;bead-perimeter_outer
$VEL.CP=1
LIN {X -65.721,Y -278.478,Z 40.000,A 0.000,B 0.000,C 180.000,E1 0.000} C_DIS
LIN {X -51.297,Y -281.492,Z 40.000,A 0.000,B 0.000,C 180.000,E1 0.000} C_DIS
LIN {X -36.738,Y -283.759,Z 40.000,A 0.000,B 0.000,C 180.000,E1 0.000} C_DIS
LIN {X -22.082,Y -285.274,Z 40.000,A 0.000,B 0.000,C 180.000,E1 0.000} C_DIS
LIN {X -7.367,Y -286.033,Z 40.000,A 0.000,B 0.000,C 180.000,E1 0.000} C_DIS
LIN {X 7.367,Y -286.033,Z 40.000,A 0.000,B 0.000,C 180.000,E1 0.000} C_DIS
LIN {X 16.843,Y -285.545,Z 40.000,A 0.000,B 0.000,C 180.000,E1 0.000} C_DIS
LIN {X 22.082,Y -285.274,Z 40.000,A 0.000,B 0.000,C 180.000,E1 0.000} C_DIS
LIN {X 36.738,Y -283.759,Z 40.000,A 0.000,B 0.000,C 180.000,E1 0.000} C_DIS
LIN {X 51.297,Y -281.492,Z 40.000,A 0.000,B 0.000,C 180.000,E1 0.000} C_DIS
LIN {X 65.721,Y -278.478,Z 40.000,A 0.000,B 0.000,C 180.000,E1 0.000} C_DIS
LIN {X 79.969,Y -274.726,Z 40.000,A 0.000,B 0.000,C 180.000,E1 0.000} C_DIS
LIN {X 94.005,Y -270.245,Z 40.000,A 0.000,B 0.000,C 180.000,E1 0.000} C_DIS
LIN {X 107.792,Y -265.047,Z 40.000,A 0.000,B 0.000,C 180.000,E1 0.000} C_DIS
LIN {X 121.294,Y -259.146,Z 40.000,A 0.000,B 0.000,C 180.000,E1 0.000} C_DIS
LIN {X 134.474,Y -252.559,Z 40.000,A 0.000,B 0.000,C 180.000,E1 0.000} C_DIS
LIN {X 147.297,Y -245.302,Z 40.000,A 0.000,B 0.000,C 180.000,E1 0.000} C_DIS
LIN {X 159.730,Y -237.393,Z 40.000,A 0.000,B 0.000,C 180.000,E1 0.000} C_DIS
LIN {X 171.739,Y -228.857,Z 40.000,A 0.000,B 0.000,C 180.000,E1 0.000} C_DIS
LIN {X 183.292,Y -219.713,Z 40.000,A 0.000,B 0.000,C 180.000,E1 0.000} C_DIS
LIN {X 194.358,Y -209.985,Z 40.000,A 0.000,B 0.000,C 180.000,E1 0.000} C_DIS
LIN {X 204.911,Y -199.701,Z 40.000,A 0.000,B 0.000,C 180.000,E1 0.000} C_DIS
LIN {X 214.920,Y -188.888,Z 40.000,A 0.000,B 0.000,C 180.000,E1 0.000} C_DIS
LIN {X 224.358,Y -177.574,Z 40.000,A 0.000,B 0.000,C 180.000,E1 0.000} C_DIS
LIN {X 233.202,Y -165.788,Z 40.000,A 0.000,B 0.000,C 180.000,E1 0.000} C_DIS
LIN {X 241.428,Y -153.563,Z 40.000,A 0.000,B 0.000,C 180.000,E1 0.000} C_DIS
LIN {X 249.014,Y -140.932,Z 40.000,A 0.000,B 0.000,C 180.000,E1 0.000} C_DIS
LIN {X 255.938,Y -127.926,Z 40.000,A 0.000,B 0.000,C 180.000,E1 0.000} C_DIS
LIN {X 262.185,Y -114.581,Z 40.000,A 0.000,B 0.000,C 180.000,E1 0.000} C_DIS
LIN {X 267.735,Y -100.933,Z 40.000,A 0.000,B 0.000,C 180.000,E1 0.000} C_DIS
LIN {X 272.575,Y -87.015,Z 40.000,A 0.000,B 0.000,C 180.000,E1 0.000} C_DIS
LIN {X 276.694,Y -72.868,Z 40.000,A 0.000,B 0.000,C 180.000,E1 0.000} C_DIS
LIN {X 280.078,Y -58.528,Z 40.000,A 0.000,B 0.000,C 180.000,E1 0.000} C_DIS
LIN {X 282.720,Y -44.032,Z 40.000,A 0.000,B 0.000,C 180.000,E1 0.000} C_DIS
LIN {X 284.612,Y -29.420,Z 40.000,A 0.000,B 0.000,C 180.000,E1 0.000} C_DIS
LIN {X 285.749,Y -14.730,Z 40.000,A 0.000,B 0.000,C 180.000,E1 0.000} C_DIS
LIN {X 286.128,Y 0.000,Z 40.000,A 0.000,B 0.000,C 180.000,E1 0.000} C_DIS
LIN {X 285.749,Y 14.730,Z 40.000,A 0.000,B 0.000,C 180.000,E1 0.000} C_DIS
LIN {X 284.612,Y 29.420,Z 40.000,A 0.000,B 0.000,C 180.000,E1 0.000} C_DIS
LIN {X 282.720,Y 44.032,Z 40.000,A 0.000,B 0.000,C 180.000,E1 0.000} C_DIS
LIN {X 280.078,Y 58.528,Z 40.000,A 0.000,B 0.000,C 180.000,E1 0.000} C_DIS
LIN {X 276.694,Y 72.868,Z 40.000,A 0.000,B 0.000,C 180.000,E1 0.000} C_DIS
LIN {X 272.575,Y 87.015,Z 40.000,A 0.000,B 0.000,C 180.000,E1 0.000} C_DIS
LIN {X 267.735,Y 100.932,Z 40.000,A 0.000,B 0.000,C 180.000,E1 0.000} C_DIS
LIN {X 262.185,Y 114.581,Z 40.000,A 0.000,B 0.000,C 180.000,E1 0.000} C_DIS
LIN {X 255.938,Y 127.926,Z 40.000,A 0.000,B 0.000,C 180.000,E1 0.000} C_DIS
LIN {X 249.014,Y 140.932,Z 40.000,A 0.000,B 0.000,C 180.000,E1 0.000} C_DIS
LIN {X 241.428,Y 153.563,Z 40.000,A 0.000,B 0.000,C 180.000,E1 0.000} C_DIS
LIN {X 233.202,Y 165.788,Z 40.000,A 0.000,B 0.000,C 180.000,E1 0.000} C_DIS
LIN {X 224.358,Y 177.574,Z 40.000,A 0.000,B 0.000,C 180.000,E1 0.000} C_DIS
LIN {X 214.920,Y 188.888,Z 40.000,A 0.000,B 0.000,C 180.000,E1 0.000} C_DIS
LIN {X 204.911,Y 199.701,Z 40.000,A 0.000,B 0.000,C 180.000,E1 0.000} C_DIS
LIN {X 194.358,Y 209.985,Z 40.000,A 0.000,B 0.000,C 180.000,E1 0.000} C_DIS
LIN {X 183.292,Y 219.713,Z 40.000,A 0.000,B 0.000,C 180.000,E1 0.000} C_DIS
LIN {X 171.739,Y 228.857,Z 40.000,A 0.000,B 0.000,C 180.000,E1 0.000} C_DIS
LIN {X 159.730,Y 237.393,Z 40.000,A 0.000,B 0.000,C 180.000,E1 0.000} C_DIS
LIN {X 147.297,Y 245.302,Z 40.000,A 0.000,B 0.000,C 180.000,E1 0.000} C_DIS
LIN {X 134.474,Y 252.559,Z 40.000,A 0.000,B 0.000,C 180.000,E1 0.000} C_DIS
LIN {X 121.294,Y 259.146,Z 40.000,A 0.000,B 0.000,C 180.000,E1 0.000} C_DIS
LIN {X 107.792,Y 265.047,Z 40.000,A 0.000,B 0.000,C 180.000,E1 0.000} C_DIS
LIN {X 94.005,Y 270.245,Z 40.000,A 0.000,B 0.000,C 180.000,E1 0.000} C_DIS
LIN {X 79.969,Y 274.726,Z 40.000,A 0.000,B 0.000,C 180.000,E1 0.000} C_DIS
LIN {X 65.721,Y 278.478,Z 40.000,A 0.000,B 0.000,C 180.000,E1 0.000} C_DIS
LIN {X 51.297,Y 281.492,Z 40.000,A 0.000,B 0.000,C 180.000,E1 0.000} C_DIS
LIN {X 36.738,Y 283.759,Z 40.000,A 0.000,B 0.000,C 180.000,E1 0.000} C_DIS
LIN {X 22.082,Y 285.274,Z 40.000,A 0.000,B 0.000,C 180.000,E1 0.000} C_DIS
LIN {X 7.367,Y 286.033,Z 40.000,A 0.000,B 0.000,C 180.000,E1 0.000} C_DIS
LIN {X -7.367,Y 286.033,Z 40.000,A 0.000,B 0.000,C 180.000,E1 0.000} C_DIS
LIN {X -22.082,Y 285.274,Z 40.000,A 0.000,B 0.000,C 180.000,E1 0.000} C_DIS
LIN {X -36.738,Y 283.759,Z 40.000,A 0.000,B 0.000,C 180.000,E1 0.000} C_DIS
LIN {X -51.297,Y 281.492,Z 40.000,A 0.000,B 0.000,C 180.000,E1 0.000} C_DIS
LIN {X -65.721,Y 278.478,Z 40.000,A 0.000,B 0.000,C 180.000,E1 0.000} C_DIS
LIN {X -79.969,Y 274.726,Z 40.000,A 0.000,B 0.000,C 180.000,E1 0.000} C_DIS
LIN {X -94.005,Y 270.245,Z 40.000,A 0.000,B 0.000,C 180.000,E1 0.000} C_DIS
LIN {X -107.792,Y 265.047,Z 40.000,A 0.000,B 0.000,C 180.000,E1 0.000} C_DIS
LIN {X -121.294,Y 259.146,Z 40.000,A 0.000,B 0.000,C 180.000,E1 0.000} C_DIS
LIN {X -134.474,Y 252.559,Z 40.000,A 0.000,B 0.000,C 180.000,E1 0.000} C_DIS
LIN {X -147.297,Y 245.302,Z 40.000,A 0.000,B 0.000,C 180.000,E1 0.000} C_DIS
LIN {X -159.730,Y 237.393,Z 40.000,A 0.000,B 0.000,C 180.000,E1 0.000} C_DIS
LIN {X -171.739,Y 228.857,Z 40.000,A 0.000,B 0.000,C 180.000,E1 0.000} C_DIS
LIN {X -183.292,Y 219.713,Z 40.000,A 0.000,B 0.000,C 180.000,E1 0.000} C_DIS
LIN {X -194.358,Y 209.985,Z 40.000,A 0.000,B 0.000,C 180.000,E1 0.000} C_DIS
LIN {X -204.911,Y 199.701,Z 40.000,A 0.000,B 0.000,C 180.000,E1 0.000} C_DIS
LIN {X -214.920,Y 188.888,Z 40.000,A 0.000,B 0.000,C 180.000,E1 0.000} C_DIS
LIN {X -224.358,Y 177.574,Z 40.000,A 0.000,B 0.000,C 180.000,E1 0.000} C_DIS
LIN {X -233.202,Y 165.788,Z 40.000,A 0.000,B 0.000,C 180.000,E1 0.000} C_DIS
LIN {X -241.428,Y 153.563,Z 40.000,A 0.000,B 0.000,C 180.000,E1 0.000} C_DIS
LIN {X -249.014,Y 140.932,Z 40.000,A 0.000,B 0.000,C 180.000,E1 0.000} C_DIS
LIN {X -255.938,Y 127.926,Z 40.000,A 0.000,B 0.000,C 180.000,E1 0.000} C_DIS
LIN {X -262.185,Y 114.581,Z 40.000,A 0.000,B 0.000,C 180.000,E1 0.000} C_DIS
LIN {X -267.735,Y 100.933,Z 40.000,A 0.000,B 0.000,C 180.000,E1 0.000} C_DIS
LIN {X -272.575,Y 87.015,Z 40.000,A 0.000,B 0.000,C 180.000,E1 0.000} C_DIS
LIN {X -276.694,Y 72.868,Z 40.000,A 0.000,B 0.000,C 180.000,E1 0.000} C_DIS
LIN {X -280.078,Y 58.528,Z 40.000,A 0.000,B 0.000,C 180.000,E1 0.000} C_DIS
LIN {X -282.720,Y 44.032,Z 40.000,A 0.000,B 0.000,C 180.000,E1 0.000} C_DIS
LIN {X -284.612,Y 29.420,Z 40.000,A 0.000,B 0.000,C 180.000,E1 0.000} C_DIS
LIN {X -285.749,Y 14.730,Z 40.000,A 0.000,B 0.000,C 180.000,E1 0.000} C_DIS
LIN {X -286.128,Y 0.000,Z 40.000,A 0.000,B 0.000,C 180.000,E1 0.000} C_DIS
LIN {X -285.749,Y -14.730,Z 40.000,A 0.000,B 0.000,C 180.000,E1 0.000} C_DIS
LIN {X -284.612,Y -29.420,Z 40.000,A 0.000,B 0.000,C 180.000,E1 0.000} C_DIS
LIN {X -282.720,Y -44.032,Z 40.000,A 0.000,B 0.000,C 180.000,E1 0.000} C_DIS
LIN {X -280.078,Y -58.528,Z 40.000,A 0.000,B 0.000,C 180.000,E1 0.000} C_DIS
LIN {X -276.694,Y -72.868,Z 40.000,A 0.000,B 0.000,C 180.000,E1 0.000} C_DIS
LIN {X -272.575,Y -87.015,Z 40.000,A 0.000,B 0.000,C 180.000,E1 0.000} C_DIS
LIN {X -269.459,Y -95.976,Z 40.000,A 0.000,B 0.000,C 180.000,E1 0.000} C_DIS
LIN {X -267.735,Y -100.932,Z 40.000,A 0.000,B 0.000,C 180.000,E1 0.000} C_DIS
LIN {X -262.185,Y -114.581,Z 40.000,A 0.000,B 0.000,C 180.000,E1 0.000} C_DIS
LIN {X -255.938,Y -127.926,Z 40.000,A 0.000,B 0.000,C 180.000,E1 0.000} C_DIS
LIN {X -249.014,Y -140.932,Z 40.000,A 0.000,B 0.000,C 180.000,E1 0.000} C_DIS
LIN {X -241.428,Y -153.563,Z 40.000,A 0.000,B 0.000,C 180.000,E1 0.000} C_DIS
LIN {X -233.202,Y -165.788,Z 40.000,A 0.000,B 0.000,C 180.000,E1 0.000} C_DIS
LIN {X -224.358,Y -177.574,Z 40.000,A 0.000,B 0.000,C 180.000,E1 0.000} C_DIS
LIN {X -214.920,Y -188.888,Z 40.000,A 0.000,B 0.000,C 180.000,E1 0.000} C_DIS
LIN {X -204.911,Y -199.701,Z 40.000,A 0.000,B 0.000,C 180.000,E1 0.000} C_DIS
LIN {X -194.358,Y -209.985,Z 40.000,A 0.000,B 0.000,C 180.000,E1 0.000} C_DIS
LIN {X -183.292,Y -219.713,Z 40.000,A 0.000,B 0.000,C 180.000,E1 0.000} C_DIS
LIN {X -171.739,Y -228.857,Z 40.000,A 0.000,B 0.000,C 180.000,E1 0.000} C_DIS
LIN {X -159.730,Y -237.393,Z 40.000,A 0.000,B 0.000,C 180.000,E1 0.000} C_DIS
LIN {X -147.297,Y -245.302,Z 40.000,A 0.000,B 0.000,C 180.000,E1 0.000} C_DIS
LIN {X -134.474,Y -252.559,Z 40.000,A 0.000,B 0.000,C 180.000,E1 0.000} C_DIS
LIN {X -121.294,Y -259.146,Z 40.000,A 0.000,B 0.000,C 180.000,E1 0.000} C_DIS
LIN {X -107.792,Y -265.047,Z 40.000,A 0.000,B 0.000,C 180.000,E1 0.000} C_DIS
LIN {X -94.005,Y -270.245,Z 40.000,A 0.000,B 0.000,C 180.000,E1 0.000} C_DIS
LIN {X -79.969,Y -274.726,Z 40.000,A 0.000,B 0.000,C 180.000,E1 0.000} C_DIS
;rapid-leaky
$VEL.CP=0.3
LIN {X -75.624,Y -259.800,Z 40.000,A 0.000,B 0.000,C 180.000,E1 0.000} C_DIS
;bead-perimeter_inner
$VEL.CP=1
LIN {X -62.150,Y -263.349,Z 40.000,A 0.000,B 0.000,C 180.000,E1 0.000} C_DIS
LIN {X -48.511,Y -266.199,Z 40.000,A 0.000,B 0.000,C 180.000,E1 0.000} C_DIS
LIN {X -34.743,Y -268.343,Z 40.000,A 0.000,B 0.000,C 180.000,E1 0.000} C_DIS
LIN {X -20.882,Y -269.776,Z 40.000,A 0.000,B 0.000,C 180.000,E1 0.000} C_DIS
LIN {X -6.967,Y -270.493,Z 40.000,A 0.000,B 0.000,C 180.000,E1 0.000} C_DIS
LIN {X 6.967,Y -270.493,Z 40.000,A 0.000,B 0.000,C 180.000,E1 0.000} C_DIS
LIN {X 16.043,Y -270.025,Z 40.000,A 0.000,B 0.000,C 180.000,E1 0.000} C_DIS
LIN {X 20.882,Y -269.776,Z 40.000,A 0.000,B 0.000,C 180.000,E1 0.000} C_DIS
LIN {X 34.743,Y -268.343,Z 40.000,A 0.000,B 0.000,C 180.000,E1 0.000} C_DIS
LIN {X 48.511,Y -266.199,Z 40.000,A 0.000,B 0.000,C 180.000,E1 0.000} C_DIS
LIN {X 62.150,Y -263.349,Z 40.000,A 0.000,B 0.000,C 180.000,E1 0.000} C_DIS
LIN {X 75.624,Y -259.800,Z 40.000,A 0.000,B 0.000,C 180.000,E1 0.000} C_DIS
LIN {X 88.898,Y -255.563,Z 40.000,A 0.000,B 0.000,C 180.000,E1 0.000} C_DIS
LIN {X 101.936,Y -250.648,Z 40.000,A 0.000,B 0.000,C 180.000,E1 0.000} C_DIS
LIN {X 114.704,Y -245.067,Z 40.000,A 0.000,B 0.000,C 180.000,E1 0.000} C_DIS
LIN {X 127.168,Y -238.838,Z 40.000,A 0.000,B 0.000,C 180.000,E1 0.000} C_DIS
LIN {X 139.294,Y -231.975,Z 40.000,A 0.000,B 0.000,C 180.000,E1 0.000} C_DIS
LIN {X 151.052,Y -224.496,Z 40.000,A 0.000,B 0.000,C 180.000,E1 0.000} C_DIS
LIN {X 162.409,Y -216.423,Z 40.000,A 0.000,B 0.000,C 180.000,E1 0.000} C_DIS
LIN {X 173.333,Y -207.776,Z 40.000,A 0.000,B 0.000,C 180.000,E1 0.000} C_DIS
LIN {X 183.799,Y -198.577,Z 40.000,A 0.000,B 0.000,C 180.000,E1 0.000} C_DIS
LIN {X 193.778,Y -188.852,Z 40.000,A 0.000,B 0.000,C 180.000,E1 0.000} C_DIS
LIN {X 203.243,Y -178.626,Z 40.000,A 0.000,B 0.000,C 180.000,E1 0.000} C_DIS
LIN {X 212.169,Y -167.927,Z 40.000,A 0.000,B 0.000,C 180.000,E1 0.000} C_DIS
LIN {X 220.533,Y -156.781,Z 40.000,A 0.000,B 0.000,C 180.000,E1 0.000} C_DIS
LIN {X 228.312,Y -145.220,Z 40.000,A 0.000,B 0.000,C 180.000,E1 0.000} C_DIS
LIN {X 235.485,Y -133.275,Z 40.000,A 0.000,B 0.000,C 180.000,E1 0.000} C_DIS
LIN {X 242.033,Y -120.975,Z 40.000,A 0.000,B 0.000,C 180.000,E1 0.000} C_DIS
LIN {X 247.940,Y -108.356,Z 40.000,A 0.000,B 0.000,C 180.000,E1 0.000} C_DIS
LIN {X 253.189,Y -95.450,Z 40.000,A 0.000,B 0.000,C 180.000,E1 0.000} C_DIS
LIN {X 257.767,Y -82.287,Z 40.000,A 0.000,B 0.000,C 180.000,E1 0.000} C_DIS
LIN {X 261.662,Y -68.909,Z 40.000,A 0.000,B 0.000,C 180.000,E1 0.000} C_DIS
LIN {X 264.862,Y -55.348,Z 40.000,A 0.000,B 0.000,C 180.000,E1 0.000} C_DIS
LIN {X 267.360,Y -41.639,Z 40.000,A 0.000,B 0.000,C 180.000,E1 0.000} C_DIS
LIN {X 269.149,Y -27.822,Z 40.000,A 0.000,B 0.000,C 180.000,E1 0.000} C_DIS
LIN {X 270.224,Y -13.929,Z 40.000,A 0.000,B 0.000,C 180.000,E1 0.000} C_DIS
LIN {X 270.583,Y 0.000,Z 40.000,A 0.000,B 0.000,C 180.000,E1 0.000} C_DIS
LIN {X 270.224,Y 13.929,Z 40.000,A 0.000,B 0.000,C 180.000,E1 0.000} C_DIS
LIN {X 269.149,Y 27.822,Z 40.000,A 0.000,B 0.000,C 180.000,E1 0.000} C_DIS
LIN {X 267.360,Y 41.639,Z 40.000,A 0.000,B 0.000,C 180.000,E1 0.000} C_DIS
LIN {X 264.862,Y 55.348,Z 40.000,A 0.000,B 0.000,C 180.000,E1 0.000} C_DIS
LIN {X 261.662,Y 68.909,Z 40.000,A 0.000,B 0.000,C 180.000,E1 0.000} C_DIS
LIN {X 257.766,Y 82.288,Z 40.000,A 0.000,B 0.000,C 180.000,E1 0.000} C_DIS
LIN {X 253.189,Y 95.449,Z 40.000,A 0.000,B 0.000,C 180.000,E1 0.000} C_DIS
LIN {X 247.940,Y 108.356,Z 40.000,A 0.000,B 0.000,C 180.000,E1 0.000} C_DIS
LIN {X 242.033,Y 120.975,Z 40.000,A 0.000,B 0.000,C 180.000,E1 0.000} C_DIS
LIN {X 235.485,Y 133.275,Z 40.000,A 0.000,B 0.000,C 180.000,E1 0.000} C_DIS
LIN {X 228.312,Y 145.220,Z 40.000,A 0.000,B 0.000,C 180.000,E1 0.000} C_DIS
LIN {X 220.533,Y 156.781,Z 40.000,A 0.000,B 0.000,C 180.000,E1 0.000} C_DIS
LIN {X 212.169,Y 167.927,Z 40.000,A 0.000,B 0.000,C 180.000,E1 0.000} C_DIS
LIN {X 203.243,Y 178.626,Z 40.000,A 0.000,B 0.000,C 180.000,E1 0.000} C_DIS
LIN {X 193.778,Y 188.852,Z 40.000,A 0.000,B 0.000,C 180.000,E1 0.000} C_DIS
LIN {X 183.799,Y 198.577,Z 40.000,A 0.000,B 0.000,C 180.000,E1 0.000} C_DIS
LIN {X 173.333,Y 207.776,Z 40.000,A 0.000,B 0.000,C 180.000,E1 0.000} C_DIS
LIN {X 162.409,Y 216.423,Z 40.000,A 0.000,B 0.000,C 180.000,E1 0.000} C_DIS
LIN {X 151.052,Y 224.496,Z 40.000,A 0.000,B 0.000,C 180.000,E1 0.000} C_DIS
LIN {X 139.294,Y 231.975,Z 40.000,A 0.000,B 0.000,C 180.000,E1 0.000} C_DIS
LIN {X 127.168,Y 238.838,Z 40.000,A 0.000,B 0.000,C 180.000,E1 0.000} C_DIS
LIN {X 114.704,Y 245.067,Z 40.000,A 0.000,B 0.000,C 180.000,E1 0.000} C_DIS
LIN {X 101.936,Y 250.648,Z 40.000,A 0.000,B 0.000,C 180.000,E1 0.000} C_DIS
LIN {X 88.898,Y 255.563,Z 40.000,A 0.000,B 0.000,C 180.000,E1 0.000} C_DIS
LIN {X 75.624,Y 259.800,Z 40.000,A 0.000,B 0.000,C 180.000,E1 0.000} C_DIS
LIN {X 62.150,Y 263.349,Z 40.000,A 0.000,B 0.000,C 180.000,E1 0.000} C_DIS
LIN {X 48.511,Y 266.199,Z 40.000,A 0.000,B 0.000,C 180.000,E1 0.000} C_DIS
LIN {X 34.743,Y 268.343,Z 40.000,A 0.000,B 0.000,C 180.000,E1 0.000} C_DIS
LIN {X 20.882,Y 269.776,Z 40.000,A 0.000,B 0.000,C 180.000,E1 0.000} C_DIS
LIN {X 6.967,Y 270.493,Z 40.000,A 0.000,B 0.000,C 180.000,E1 0.000} C_DIS
LIN {X -6.967,Y 270.493,Z 40.000,A 0.000,B 0.000,C 180.000,E1 0.000} C_DIS
LIN {X -20.882,Y 269.776,Z 40.000,A 0.000,B 0.000,C 180.000,E1 0.000} C_DIS
LIN {X -34.743,Y 268.343,Z 40.000,A 0.000,B 0.000,C 180.000,E1 0.000} C_DIS
LIN {X -48.511,Y 266.199,Z 40.000,A 0.000,B 0.000,C 180.000,E1 0.000} C_DIS
LIN {X -62.150,Y 263.349,Z 40.000,A 0.000,B 0.000,C 180.000,E1 0.000} C_DIS
LIN {X -75.624,Y 259.800,Z 40.000,A 0.000,B 0.000,C 180.000,E1 0.000} C_DIS
LIN {X -88.898,Y 255.563,Z 40.000,A 0.000,B 0.000,C 180.000,E1 0.000} C_DIS
LIN {X -101.936,Y 250.648,Z 40.000,A 0.000,B 0.000,C 180.000,E1 0.000} C_DIS
LIN {X -114.704,Y 245.067,Z 40.000,A 0.000,B 0.000,C 180.000,E1 0.000} C_DIS
LIN {X -127.168,Y 238.838,Z 40.000,A 0.000,B 0.000,C 180.000,E1 0.000} C_DIS
LIN {X -139.294,Y 231.975,Z 40.000,A 0.000,B 0.000,C 180.000,E1 0.000} C_DIS
LIN {X -151.052,Y 224.496,Z 40.000,A 0.000,B 0.000,C 180.000,E1 0.000} C_DIS
LIN {X -162.409,Y 216.423,Z 40.000,A 0.000,B 0.000,C 180.000,E1 0.000} C_DIS
LIN {X -173.333,Y 207.776,Z 40.000,A 0.000,B 0.000,C 180.000,E1 0.000} C_DIS
LIN {X -183.799,Y 198.577,Z 40.000,A 0.000,B 0.000,C 180.000,E1 0.000} C_DIS
LIN {X -193.778,Y 188.852,Z 40.000,A 0.000,B 0.000,C 180.000,E1 0.000} C_DIS
LIN {X -203.243,Y 178.626,Z 40.000,A 0.000,B 0.000,C 180.000,E1 0.000} C_DIS
LIN {X -212.169,Y 167.927,Z 40.000,A 0.000,B 0.000,C 180.000,E1 0.000} C_DIS
LIN {X -220.533,Y 156.781,Z 40.000,A 0.000,B 0.000,C 180.000,E1 0.000} C_DIS
LIN {X -228.312,Y 145.220,Z 40.000,A 0.000,B 0.000,C 180.000,E1 0.000} C_DIS
LIN {X -235.485,Y 133.275,Z 40.000,A 0.000,B 0.000,C 180.000,E1 0.000} C_DIS
LIN {X -242.033,Y 120.975,Z 40.000,A 0.000,B 0.000,C 180.000,E1 0.000} C_DIS
LIN {X -247.940,Y 108.356,Z 40.000,A 0.000,B 0.000,C 180.000,E1 0.000} C_DIS
LIN {X -253.189,Y 95.450,Z 40.000,A 0.000,B 0.000,C 180.000,E1 0.000} C_DIS
LIN {X -257.767,Y 82.287,Z 40.000,A 0.000,B 0.000,C 180.000,E1 0.000} C_DIS
LIN {X -261.662,Y 68.909,Z 40.000,A 0.000,B 0.000,C 180.000,E1 0.000} C_DIS
LIN {X -264.862,Y 55.348,Z 40.000,A 0.000,B 0.000,C 180.000,E1 0.000} C_DIS
LIN {X -267.360,Y 41.639,Z 40.000,A 0.000,B 0.000,C 180.000,E1 0.000} C_DIS
LIN {X -269.149,Y 27.822,Z 40.000,A 0.000,B 0.000,C 180.000,E1 0.000} C_DIS
LIN {X -270.224,Y 13.929,Z 40.000,A 0.000,B 0.000,C 180.000,E1 0.000} C_DIS
LIN {X -270.583,Y 0.000,Z 40.000,A 0.000,B 0.000,C 180.000,E1 0.000} C_DIS
LIN {X -270.224,Y -13.929,Z 40.000,A 0.000,B 0.000,C 180.000,E1 0.000} C_DIS
LIN {X -269.149,Y -27.822,Z 40.000,A 0.000,B 0.000,C 180.000,E1 0.000} C_DIS
LIN {X -267.360,Y -41.639,Z 40.000,A 0.000,B 0.000,C 180.000,E1 0.000} C_DIS
LIN {X -264.862,Y -55.348,Z 40.000,A 0.000,B 0.000,C 180.000,E1 0.000} C_DIS
LIN {X -261.662,Y -68.909,Z 40.000,A 0.000,B 0.000,C 180.000,E1 0.000} C_DIS
LIN {X -257.766,Y -82.288,Z 40.000,A 0.000,B 0.000,C 180.000,E1 0.000} C_DIS
LIN {X -254.782,Y -90.870,Z 40.000,A 0.000,B 0.000,C 180.000,E1 0.000} C_DIS
LIN {X -253.189,Y -95.449,Z 40.000,A 0.000,B 0.000,C 180.000,E1 0.000} C_DIS
LIN {X -247.940,Y -108.356,Z 40.000,A 0.000,B 0.000,C 180.000,E1 0.000} C_DIS
LIN {X -242.033,Y -120.975,Z 40.000,A 0.000,B 0.000,C 180.000,E1 0.000} C_DIS
LIN {X -235.485,Y -133.275,Z 40.000,A 0.000,B 0.000,C 180.000,E1 0.000} C_DIS
LIN {X -228.312,Y -145.220,Z 40.000,A 0.000,B 0.000,C 180.000,E1 0.000} C_DIS
LIN {X -220.533,Y -156.781,Z 40.000,A 0.000,B 0.000,C 180.000,E1 0.000} C_DIS
LIN {X -212.169,Y -167.927,Z 40.000,A 0.000,B 0.000,C 180.000,E1 0.000} C_DIS
LIN {X -203.243,Y -178.626,Z 40.000,A 0.000,B 0.000,C 180.000,E1 0.000} C_DIS
LIN {X -193.778,Y -188.852,Z 40.000,A 0.000,B 0.000,C 180.000,E1 0.000} C_DIS
LIN {X -183.799,Y -198.577,Z 40.000,A 0.000,B 0.000,C 180.000,E1 0.000} C_DIS
LIN {X -173.333,Y -207.776,Z 40.000,A 0.000,B 0.000,C 180.000,E1 0.000} C_DIS
LIN {X -162.409,Y -216.423,Z 40.000,A 0.000,B 0.000,C 180.000,E1 0.000} C_DIS
LIN {X -151.052,Y -224.496,Z 40.000,A 0.000,B 0.000,C 180.000,E1 0.000} C_DIS
LIN {X -139.294,Y -231.975,Z 40.000,A 0.000,B 0.000,C 180.000,E1 0.000} C_DIS
LIN {X -127.168,Y -238.838,Z 40.000,A 0.000,B 0.000,C 180.000,E1 0.000} C_DIS
LIN {X -114.704,Y -245.067,Z 40.000,A 0.000,B 0.000,C 180.000,E1 0.000} C_DIS
LIN {X -101.936,Y -250.648,Z 40.000,A 0.000,B 0.000,C 180.000,E1 0.000} C_DIS
LIN {X -88.898,Y -255.563,Z 40.000,A 0.000,B 0.000,C 180.000,E1 0.000} C_DIS
LIN {X -75.624,Y -259.800,Z 40.000,A 0.000,B 0.000,C 180.000,E1 0.000} C_DIS
$VEL.CP=0.3
LIN {X -75.624,Y -259.800,Z 40.000,A 0.000,B 0.000,C 180.000,E1 0.000} C_DIS

EXTRUDER_STATE=FALSE

LIN {X 316.392,Y -180.278,Z 440.000,A 0.000,B 0.000,C 180.000,E1 0.000} C_DIS
LIN {X 126.528,Y -218.793,Z 440.000,A 0.000,B 0.000,C 180.000,E1 0.000} C_DIS
LIN {X 126.528,Y -218.793,Z 40.000,A 0.000,B 0.000,C 180.000,E1 0.000} C_DIS
LIN {X 126.528,Y -218.793,Z 40.000,A 0.000,B 0.000,C 180.000,E1 0.000} C_DIS
EXTRUDER_STATE=TRUE

;bead-solid_infill
$VEL.CP=1
LIN {X 218.862,Y -126.458,Z 40.000,A 0.000,B 0.000,C 180.000,E1 0.000} C_DIS
LIN {X 220.023,Y -124.525,Z 40.000,A 0.000,B 0.000,C 180.000,E1 0.000} C_DIS
LIN {X 222.894,Y -119.132,Z 40.000,A 0.000,B 0.000,C 180.000,E1 0.000} C_DIS
LIN {X 226.142,Y -113.032,Z 40.000,A 0.000,B 0.000,C 180.000,E1 0.000} C_DIS
LIN {X 231.661,Y -101.241,Z 40.000,A 0.000,B 0.000,C 180.000,E1 0.000} C_DIS
LIN {X 236.565,Y -89.183,Z 40.000,A 0.000,B 0.000,C 180.000,E1 0.000} C_DIS
LIN {X 240.842,Y -76.884,Z 40.000,A 0.000,B 0.000,C 180.000,E1 0.000} C_DIS
LIN {X 242.404,Y -71.521,Z 40.000,A 0.000,B 0.000,C 180.000,E1 0.000} C_DIS
LIN {X 71.429,Y -242.496,Z 40.000,A 0.000,B 0.000,C 180.000,E1 0.000} C_DIS
LIN {X 70.658,Y -242.742,Z 40.000,A 0.000,B 0.000,C 180.000,E1 0.000} C_DIS
LIN {X 58.069,Y -246.058,Z 40.000,A 0.000,B 0.000,C 180.000,E1 0.000} C_DIS
LIN {X 45.326,Y -248.721,Z 40.000,A 0.000,B 0.000,C 180.000,E1 0.000} C_DIS
LIN {X 32.462,Y -250.724,Z 40.000,A 0.000,B 0.000,C 180.000,E1 0.000} C_DIS
LIN {X 31.730,Y -250.800,Z 40.000,A 0.000,B 0.000,C 180.000,E1 0.000} C_DIS
LIN {X 250.725,Y -31.804,Z 40.000,A 0.000,B 0.000,C 180.000,E1 0.000} C_DIS
LIN {X 251.478,Y -25.994,Z 40.000,A 0.000,B 0.000,C 180.000,E1 0.000} C_DIS
LIN {X 252.482,Y -13.015,Z 40.000,A 0.000,B 0.000,C 180.000,E1 0.000} C_DIS
LIN {X 252.817,Y 0.000,Z 40.000,A 0.000,B 0.000,C 180.000,E1 0.000} C_DIS
LIN {X 252.775,Y 1.641,Z 40.000,A 0.000,B 0.000,C 180.000,E1 0.000} C_DIS
LIN {X -1.599,Y -252.733,Z 40.000,A 0.000,B 0.000,C 180.000,E1 0.000} C_DIS
LIN {X -6.509,Y -252.733,Z 40.000,A 0.000,B 0.000,C 180.000,E1 0.000} C_DIS
LIN {X -19.511,Y -252.063,Z 40.000,A 0.000,B 0.000,C 180.000,E1 0.000} C_DIS
LIN {X -31.124,Y -250.862,Z 40.000,A 0.000,B 0.000,C 180.000,E1 0.000} C_DIS
LIN {X 250.819,Y 31.081,Z 40.000,A 0.000,B 0.000,C 180.000,E1 0.000} C_DIS
LIN {X 249.806,Y 38.905,Z 40.000,A 0.000,B 0.000,C 180.000,E1 0.000} C_DIS
LIN {X 247.471,Y 51.715,Z 40.000,A 0.000,B 0.000,C 180.000,E1 0.000} C_DIS
LIN {X 246.056,Y 57.713,Z 40.000,A 0.000,B 0.000,C 180.000,E1 0.000} C_DIS
LIN {X -57.776,Y -246.119,Z 40.000,A 0.000,B 0.000,C 180.000,E1 0.000} C_DIS
LIN {X -58.069,Y -246.058,Z 40.000,A 0.000,B 0.000,C 180.000,E1 0.000} C_DIS
LIN {X -70.658,Y -242.742,Z 40.000,A 0.000,B 0.000,C 180.000,E1 0.000} C_DIS
LIN {X -82.132,Y -239.079,Z 40.000,A 0.000,B 0.000,C 180.000,E1 0.000} C_DIS
LIN {X 239.033,Y 82.086,Z 40.000,A 0.000,B 0.000,C 180.000,E1 0.000} C_DIS
LIN {X 236.565,Y 89.182,Z 40.000,A 0.000,B 0.000,C 180.000,E1 0.000} C_DIS
LIN {X 231.661,Y 101.241,Z 40.000,A 0.000,B 0.000,C 180.000,E1 0.000} C_DIS
LIN {X 230.109,Y 104.557,Z 40.000,A 0.000,B 0.000,C 180.000,E1 0.000} C_DIS
LIN {X -104.565,Y -230.117,Z 40.000,A 0.000,B 0.000,C 180.000,E1 0.000} C_DIS
LIN {X -107.173,Y -228.977,Z 40.000,A 0.000,B 0.000,C 180.000,E1 0.000} C_DIS
LIN {X -118.819,Y -223.156,Z 40.000,A 0.000,B 0.000,C 180.000,E1 0.000} C_DIS
LIN {X -125.320,Y -219.476,Z 40.000,A 0.000,B 0.000,C 180.000,E1 0.000} C_DIS
LIN {X 219.520,Y 125.364,Z 40.000,A 0.000,B 0.000,C 180.000,E1 0.000} C_DIS
LIN {X 213.322,Y 135.685,Z 40.000,A 0.000,B 0.000,C 180.000,E1 0.000} C_DIS
LIN {X 207.338,Y 144.577,Z 40.000,A 0.000,B 0.000,C 180.000,E1 0.000} C_DIS
LIN {X -144.560,Y -207.321,Z 40.000,A 0.000,B 0.000,C 180.000,E1 0.000} C_DIS
LIN {X -151.746,Y -202.213,Z 40.000,A 0.000,B 0.000,C 180.000,E1 0.000} C_DIS
LIN {X -161.952,Y -194.135,Z 40.000,A 0.000,B 0.000,C 180.000,E1 0.000} C_DIS
LIN {X -162.387,Y -193.752,Z 40.000,A 0.000,B 0.000,C 180.000,E1 0.000} C_DIS
LIN {X 193.703,Y 162.338,Z 40.000,A 0.000,B 0.000,C 180.000,E1 0.000} C_DIS
LIN {X 189.899,Y 166.897,Z 40.000,A 0.000,B 0.000,C 180.000,E1 0.000} C_DIS
LIN {X 181.055,Y 176.452,Z 40.000,A 0.000,B 0.000,C 180.000,E1 0.000} C_DIS
LIN {X 178.708,Y 178.739,Z 40.000,A 0.000,B 0.000,C 180.000,E1 0.000} C_DIS
LIN {X -178.739,Y -178.709,Z 40.000,A 0.000,B 0.000,C 180.000,E1 0.000} C_DIS
LIN {X -181.055,Y -176.452,Z 40.000,A 0.000,B 0.000,C 180.000,E1 0.000} C_DIS
LIN {X -189.899,Y -166.897,Z 40.000,A 0.000,B 0.000,C 180.000,E1 0.000} C_DIS
LIN {X -193.730,Y -162.305,Z 40.000,A 0.000,B 0.000,C 180.000,E1 0.000} C_DIS
LIN {X 162.355,Y 193.781,Z 40.000,A 0.000,B 0.000,C 180.000,E1 0.000} C_DIS
LIN {X 161.952,Y 194.135,Z 40.000,A 0.000,B 0.000,C 180.000,E1 0.000} C_DIS
LIN {X 151.746,Y 202.213,Z 40.000,A 0.000,B 0.000,C 180.000,E1 0.000} C_DIS
LIN {X 144.524,Y 207.346,Z 40.000,A 0.000,B 0.000,C 180.000,E1 0.000} C_DIS
LIN {X -207.362,Y -144.541,Z 40.000,A 0.000,B 0.000,C 180.000,E1 0.000} C_DIS
LIN {X -213.322,Y -135.685,Z 40.000,A 0.000,B 0.000,C 180.000,E1 0.000} C_DIS
LIN {X -219.542,Y -125.326,Z 40.000,A 0.000,B 0.000,C 180.000,E1 0.000} C_DIS
LIN {X 125.281,Y 219.498,Z 40.000,A 0.000,B 0.000,C 180.000,E1 0.000} C_DIS
LIN {X 118.819,Y 223.156,Z 40.000,A 0.000,B 0.000,C 180.000,E1 0.000} C_DIS
LIN {X 107.173,Y 228.977,Z 40.000,A 0.000,B 0.000,C 180.000,E1 0.000} C_DIS
LIN {X 104.522,Y 230.135,Z 40.000,A 0.000,B 0.000,C 180.000,E1 0.000} C_DIS
LIN {X -230.128,Y -104.516,Z 40.000,A 0.000,B 0.000,C 180.000,E1 0.000} C_DIS
LIN {X -231.661,Y -101.241,Z 40.000,A 0.000,B 0.000,C 180.000,E1 0.000} C_DIS
LIN {X -236.565,Y -89.182,Z 40.000,A 0.000,B 0.000,C 180.000,E1 0.000} C_DIS
LIN {X -237.953,Y -85.193,Z 40.000,A 0.000,B 0.000,C 180.000,E1 0.000} C_DIS
LIN {X -239.049,Y -82.041,Z 40.000,A 0.000,B 0.000,C 180.000,E1 0.000} C_DIS
LIN {X 82.086,Y 239.094,Z 40.000,A 0.000,B 0.000,C 180.000,E1 0.000} C_DIS
LIN {X 70.658,Y 242.742,Z 40.000,A 0.000,B 0.000,C 180.000,E1 0.000} C_DIS
LIN {X 58.069,Y 246.058,Z 40.000,A 0.000,B 0.000,C 180.000,E1 0.000} C_DIS
LIN {X 57.726,Y 246.130,Z 40.000,A 0.000,B 0.000,C 180.000,E1 0.000} C_DIS
LIN {X -246.067,Y -57.664,Z 40.000,A 0.000,B 0.000,C 180.000,E1 0.000} C_DIS
LIN {X -247.471,Y -51.715,Z 40.000,A 0.000,B 0.000,C 180.000,E1 0.000} C_DIS
LIN {X -249.806,Y -38.905,Z 40.000,A 0.000,B 0.000,C 180.000,E1 0.000} C_DIS
LIN {X -250.826,Y -31.027,Z 40.000,A 0.000,B 0.000,C 180.000,E1 0.000} C_DIS
LIN {X 31.069,Y 250.868,Z 40.000,A 0.000,B 0.000,C 180.000,E1 0.000} C_DIS
LIN {X 19.511,Y 252.063,Z 40.000,A 0.000,B 0.000,C 180.000,E1 0.000} C_DIS
LIN {X 6.509,Y 252.733,Z 40.000,A 0.000,B 0.000,C 180.000,E1 0.000} C_DIS
LIN {X 1.538,Y 252.733,Z 40.000,A 0.000,B 0.000,C 180.000,E1 0.000} C_DIS
LIN {X -252.777,Y -1.582,Z 40.000,A 0.000,B 0.000,C 180.000,E1 0.000} C_DIS
LIN {X -252.817,Y 0.000,Z 40.000,A 0.000,B 0.000,C 180.000,E1 0.000} C_DIS
LIN {X -252.482,Y 13.015,Z 40.000,A 0.000,B 0.000,C 180.000,E1 0.000} C_DIS
LIN {X -251.478,Y 25.994,Z 40.000,A 0.000,B 0.000,C 180.000,E1 0.000} C_DIS
LIN {X -250.716,Y 31.874,Z 40.000,A 0.000,B 0.000,C 180.000,E1 0.000} C_DIS
LIN {X -31.798,Y 250.793,Z 40.000,A 0.000,B 0.000,C 180.000,E1 0.000} C_DIS
LIN {X -32.462,Y 250.724,Z 40.000,A 0.000,B 0.000,C 180.000,E1 0.000} C_DIS
LIN {X -45.326,Y 248.721,Z 40.000,A 0.000,B 0.000,C 180.000,E1 0.000} C_DIS
LIN {X -58.069,Y 246.058,Z 40.000,A 0.000,B 0.000,C 180.000,E1 0.000} C_DIS
LIN {X -70.658,Y 242.742,Z 40.000,A 0.000,B 0.000,C 180.000,E1 0.000} C_DIS
LIN {X -71.518,Y 242.468,Z 40.000,A 0.000,B 0.000,C 180.000,E1 0.000} C_DIS
LIN {X -242.379,Y 71.607,Z 40.000,A 0.000,B 0.000,C 180.000,E1 0.000} C_DIS
LIN {X -240.842,Y 76.884,Z 40.000,A 0.000,B 0.000,C 180.000,E1 0.000} C_DIS
LIN {X -236.565,Y 89.183,Z 40.000,A 0.000,B 0.000,C 180.000,E1 0.000} C_DIS
LIN {X -231.661,Y 101.241,Z 40.000,A 0.000,B 0.000,C 180.000,E1 0.000} C_DIS
LIN {X -226.142,Y 113.032,Z 40.000,A 0.000,B 0.000,C 180.000,E1 0.000} C_DIS
LIN {X -220.023,Y 124.525,Z 40.000,A 0.000,B 0.000,C 180.000,E1 0.000} C_DIS
LIN {X -218.771,Y 126.610,Z 40.000,A 0.000,B 0.000,C 180.000,E1 0.000} C_DIS
LIN {X -126.668,Y 218.714,Z 40.000,A 0.000,B 0.000,C 180.000,E1 0.000} C_DIS
;rapid-leaky
$VEL.CP=0.3
LIN {X -260.798,Y 113.975,Z 50.000,A 0.000,B 0.000,C 180.000,E1 0.000} C_DIS
;bead-perimeter_outer
$VEL.CP=0.76
LIN {X -266.319,Y 100.399,Z 50.000,A 0.000,B 0.000,C 180.000,E1 0.000} C_DIS
LIN {X -271.133,Y 86.555,Z 50.000,A 0.000,B 0.000,C 180.000,E1 0.000} C_DIS
LIN {X -275.230,Y 72.483,Z 50.000,A 0.000,B 0.000,C 180.000,E1 0.000} C_DIS
LIN {X -278.596,Y 58.219,Z 50.000,A 0.000,B 0.000,C 180.000,E1 0.000} C_DIS
LIN {X -281.224,Y 43.799,Z 50.000,A 0.000,B 0.000,C 180.000,E1 0.000} C_DIS
LIN {X -283.106,Y 29.264,Z 50.000,A 0.000,B 0.000,C 180.000,E1 0.000} C_DIS
LIN {X -284.237,Y 14.652,Z 50.000,A 0.000,B 0.000,C 180.000,E1 0.000} C_DIS
LIN {X -284.614,Y 0.000,Z 50.000,A 0.000,B 0.000,C 180.000,E1 0.000} C_DIS
LIN {X -284.237,Y -14.652,Z 50.000,A 0.000,B 0.000,C 180.000,E1 0.000} C_DIS
LIN {X -283.106,Y -29.264,Z 50.000,A 0.000,B 0.000,C 180.000,E1 0.000} C_DIS
LIN {X -281.224,Y -43.799,Z 50.000,A 0.000,B 0.000,C 180.000,E1 0.000} C_DIS
LIN {X -278.596,Y -58.219,Z 50.000,A 0.000,B 0.000,C 180.000,E1 0.000} C_DIS
LIN {X -275.230,Y -72.483,Z 50.000,A 0.000,B 0.000,C 180.000,E1 0.000} C_DIS
LIN {X -271.133,Y -86.555,Z 50.000,A 0.000,B 0.000,C 180.000,E1 0.000} C_DIS
LIN {X -266.319,Y -100.399,Z 50.000,A 0.000,B 0.000,C 180.000,E1 0.000} C_DIS
LIN {X -260.798,Y -113.975,Z 50.000,A 0.000,B 0.000,C 180.000,E1 0.000} C_DIS
LIN {X -254.584,Y -127.249,Z 50.000,A 0.000,B 0.000,C 180.000,E1 0.000} C_DIS
LIN {X -247.696,Y -140.186,Z 50.000,A 0.000,B 0.000,C 180.000,E1 0.000} C_DIS
LIN {X -240.151,Y -152.752,Z 50.000,A 0.000,B 0.000,C 180.000,E1 0.000} C_DIS
LIN {X -231.969,Y -164.911,Z 50.000,A 0.000,B 0.000,C 180.000,E1 0.000} C_DIS
LIN {X -223.171,Y -176.635,Z 50.000,A 0.000,B 0.000,C 180.000,E1 0.000} C_DIS
LIN {X -213.783,Y -187.889,Z 50.000,A 0.000,B 0.000,C 180.000,E1 0.000} C_DIS
LIN {X -203.827,Y -198.645,Z 50.000,A 0.000,B 0.000,C 180.000,E1 0.000} C_DIS
LIN {X -193.331,Y -208.874,Z 50.000,A 0.000,B 0.000,C 180.000,E1 0.000} C_DIS
LIN {X -182.322,Y -218.551,Z 50.000,A 0.000,B 0.000,C 180.000,E1 0.000} C_DIS
LIN {X -170.829,Y -227.646,Z 50.000,A 0.000,B 0.000,C 180.000,E1 0.000} C_DIS
LIN {X -158.884,Y -236.139,Z 50.000,A 0.000,B 0.000,C 180.000,E1 0.000} C_DIS
LIN {X -146.518,Y -244.004,Z 50.000,A 0.000,B 0.000,C 180.000,E1 0.000} C_DIS
LIN {X -133.763,Y -251.223,Z 50.000,A 0.000,B 0.000,C 180.000,E1 0.000} C_DIS
LIN {X -120.652,Y -257.775,Z 50.000,A 0.000,B 0.000,C 180.000,E1 0.000} C_DIS
LIN {X -107.222,Y -263.646,Z 50.000,A 0.000,B 0.000,C 180.000,E1 0.000} C_DIS
LIN {X -93.508,Y -268.816,Z 50.000,A 0.000,B 0.000,C 180.000,E1 0.000} C_DIS
LIN {X -79.546,Y -273.273,Z 50.000,A 0.000,B 0.000,C 180.000,E1 0.000} C_DIS
LIN {X -65.373,Y -277.005,Z 50.000,A 0.000,B 0.000,C 180.000,E1 0.000} C_DIS
LIN {X -51.025,Y -280.003,Z 50.000,A 0.000,B 0.000,C 180.000,E1 0.000} C_DIS
LIN {X -36.544,Y -282.259,Z 50.000,A 0.000,B 0.000,C 180.000,E1 0.000} C_DIS
LIN {X -21.966,Y -283.765,Z 50.000,A 0.000,B 0.000,C 180.000,E1 0.000} C_DIS
LIN {X -7.328,Y -284.520,Z 50.000,A 0.000,B 0.000,C 180.000,E1 0.000} C_DIS
LIN {X 7.328,Y -284.520,Z 50.000,A 0.000,B 0.000,C 180.000,E1 0.000} C_DIS
LIN {X 21.966,Y -283.765,Z 50.000,A 0.000,B 0.000,C 180.000,E1 0.000} C_DIS
LIN {X 36.544,Y -282.259,Z 50.000,A 0.000,B 0.000,C 180.000,E1 0.000} C_DIS
LIN {X 51.025,Y -280.003,Z 50.000,A 0.000,B 0.000,C 180.000,E1 0.000} C_DIS
LIN {X 65.373,Y -277.005,Z 50.000,A 0.000,B 0.000,C 180.000,E1 0.000} C_DIS
LIN {X 79.546,Y -273.273,Z 50.000,A 0.000,B 0.000,C 180.000,E1 0.000} C_DIS
LIN {X 93.508,Y -268.816,Z 50.000,A 0.000,B 0.000,C 180.000,E1 0.000} C_DIS
LIN {X 107.223,Y -263.645,Z 50.000,A 0.000,B 0.000,C 180.000,E1 0.000} C_DIS
LIN {X 111.212,Y -261.902,Z 50.000,A 0.000,B 0.000,C 180.000,E1 0.000} C_DIS
LIN {X 120.652,Y -257.776,Z 50.000,A 0.000,B 0.000,C 180.000,E1 0.000} C_DIS
LIN {X 133.763,Y -251.223,Z 50.000,A 0.000,B 0.000,C 180.000,E1 0.000} C_DIS
LIN {X 146.518,Y -244.004,Z 50.000,A 0.000,B 0.000,C 180.000,E1 0.000} C_DIS
LIN {X 158.884,Y -236.139,Z 50.000,A 0.000,B 0.000,C 180.000,E1 0.000} C_DIS
LIN {X 170.829,Y -227.646,Z 50.000,A 0.000,B 0.000,C 180.000,E1 0.000} C_DIS
LIN {X 182.322,Y -218.551,Z 50.000,A 0.000,B 0.000,C 180.000,E1 0.000} C_DIS
LIN {X 193.331,Y -208.874,Z 50.000,A 0.000,B 0.000,C 180.000,E1 0.000} C_DIS
LIN {X 203.827,Y -198.645,Z 50.000,A 0.000,B 0.000,C 180.000,E1 0.000} C_DIS
LIN {X 213.783,Y -187.889,Z 50.000,A 0.000,B 0.000,C 180.000,E1 0.000} C_DIS
LIN {X 223.171,Y -176.635,Z 50.000,A 0.000,B 0.000,C 180.000,E1 0.000} C_DIS
LIN {X 231.969,Y -164.911,Z 50.000,A 0.000,B 0.000,C 180.000,E1 0.000} C_DIS
LIN {X 240.151,Y -152.752,Z 50.000,A 0.000,B 0.000,C 180.000,E1 0.000} C_DIS
LIN {X 247.696,Y -140.186,Z 50.000,A 0.000,B 0.000,C 180.000,E1 0.000} C_DIS
LIN {X 254.584,Y -127.249,Z 50.000,A 0.000,B 0.000,C 180.000,E1 0.000} C_DIS
LIN {X 260.798,Y -113.975,Z 50.000,A 0.000,B 0.000,C 180.000,E1 0.000} C_DIS
LIN {X 266.319,Y -100.399,Z 50.000,A 0.000,B 0.000,C 180.000,E1 0.000} C_DIS
LIN {X 271.133,Y -86.555,Z 50.000,A 0.000,B 0.000,C 180.000,E1 0.000} C_DIS
LIN {X 275.230,Y -72.483,Z 50.000,A 0.000,B 0.000,C 180.000,E1 0.000} C_DIS
LIN {X 278.596,Y -58.219,Z 50.000,A 0.000,B 0.000,C 180.000,E1 0.000} C_DIS
LIN {X 281.224,Y -43.799,Z 50.000,A 0.000,B 0.000,C 180.000,E1 0.000} C_DIS
LIN {X 283.106,Y -29.264,Z 50.000,A 0.000,B 0.000,C 180.000,E1 0.000} C_DIS
LIN {X 284.237,Y -14.652,Z 50.000,A 0.000,B 0.000,C 180.000,E1 0.000} C_DIS
LIN {X 284.614,Y 0.000,Z 50.000,A 0.000,B 0.000,C 180.000,E1 0.000} C_DIS
LIN {X 284.237,Y 14.652,Z 50.000,A 0.000,B 0.000,C 180.000,E1 0.000} C_DIS
LIN {X 283.106,Y 29.264,Z 50.000,A 0.000,B 0.000,C 180.000,E1 0.000} C_DIS
LIN {X 281.224,Y 43.799,Z 50.000,A 0.000,B 0.000,C 180.000,E1 0.000} C_DIS
LIN {X 278.596,Y 58.219,Z 50.000,A 0.000,B 0.000,C 180.000,E1 0.000} C_DIS
LIN {X 275.230,Y 72.483,Z 50.000,A 0.000,B 0.000,C 180.000,E1 0.000} C_DIS
LIN {X 271.133,Y 86.555,Z 50.000,A 0.000,B 0.000,C 180.000,E1 0.000} C_DIS
LIN {X 266.319,Y 100.399,Z 50.000,A 0.000,B 0.000,C 180.000,E1 0.000} C_DIS
LIN {X 260.798,Y 113.975,Z 50.000,A 0.000,B 0.000,C 180.000,E1 0.000} C_DIS
LIN {X 254.584,Y 127.249,Z 50.000,A 0.000,B 0.000,C 180.000,E1 0.000} C_DIS
LIN {X 247.696,Y 140.186,Z 50.000,A 0.000,B 0.000,C 180.000,E1 0.000} C_DIS
LIN {X 240.151,Y 152.752,Z 50.000,A 0.000,B 0.000,C 180.000,E1 0.000} C_DIS
LIN {X 231.969,Y 164.911,Z 50.000,A 0.000,B 0.000,C 180.000,E1 0.000} C_DIS
LIN {X 223.171,Y 176.635,Z 50.000,A 0.000,B 0.000,C 180.000,E1 0.000} C_DIS
LIN {X 213.783,Y 187.889,Z 50.000,A 0.000,B 0.000,C 180.000,E1 0.000} C_DIS
LIN {X 203.827,Y 198.645,Z 50.000,A 0.000,B 0.000,C 180.000,E1 0.000} C_DIS
LIN {X 193.331,Y 208.874,Z 50.000,A 0.000,B 0.000,C 180.000,E1 0.000} C_DIS
LIN {X 182.322,Y 218.551,Z 50.000,A 0.000,B 0.000,C 180.000,E1 0.000} C_DIS
LIN {X 170.829,Y 227.646,Z 50.000,A 0.000,B 0.000,C 180.000,E1 0.000} C_DIS
LIN {X 158.884,Y 236.139,Z 50.000,A 0.000,B 0.000,C 180.000,E1 0.000} C_DIS
LIN {X 146.518,Y 244.004,Z 50.000,A 0.000,B 0.000,C 180.000,E1 0.000} C_DIS
LIN {X 133.763,Y 251.223,Z 50.000,A 0.000,B 0.000,C 180.000,E1 0.000} C_DIS
LIN {X 120.652,Y 257.775,Z 50.000,A 0.000,B 0.000,C 180.000,E1 0.000} C_DIS
LIN {X 107.222,Y 263.646,Z 50.000,A 0.000,B 0.000,C 180.000,E1 0.000} C_DIS
LIN {X 93.508,Y 268.816,Z 50.000,A 0.000,B 0.000,C 180.000,E1 0.000} C_DIS
LIN {X 79.546,Y 273.273,Z 50.000,A 0.000,B 0.000,C 180.000,E1 0.000} C_DIS
LIN {X 65.373,Y 277.005,Z 50.000,A 0.000,B 0.000,C 180.000,E1 0.000} C_DIS
LIN {X 51.025,Y 280.003,Z 50.000,A 0.000,B 0.000,C 180.000,E1 0.000} C_DIS
LIN {X 36.544,Y 282.259,Z 50.000,A 0.000,B 0.000,C 180.000,E1 0.000} C_DIS
LIN {X 21.966,Y 283.765,Z 50.000,A 0.000,B 0.000,C 180.000,E1 0.000} C_DIS
LIN {X 7.328,Y 284.520,Z 50.000,A 0.000,B 0.000,C 180.000,E1 0.000} C_DIS
LIN {X -7.328,Y 284.520,Z 50.000,A 0.000,B 0.000,C 180.000,E1 0.000} C_DIS
LIN {X -21.966,Y 283.765,Z 50.000,A 0.000,B 0.000,C 180.000,E1 0.000} C_DIS
LIN {X -36.544,Y 282.259,Z 50.000,A 0.000,B 0.000,C 180.000,E1 0.000} C_DIS
LIN {X -51.025,Y 280.003,Z 50.000,A 0.000,B 0.000,C 180.000,E1 0.000} C_DIS
LIN {X -65.373,Y 277.005,Z 50.000,A 0.000,B 0.000,C 180.000,E1 0.000} C_DIS
LIN {X -79.546,Y 273.273,Z 50.000,A 0.000,B 0.000,C 180.000,E1 0.000} C_DIS
LIN {X -93.508,Y 268.816,Z 50.000,A 0.000,B 0.000,C 180.000,E1 0.000} C_DIS
LIN {X -107.223,Y 263.645,Z 50.000,A 0.000,B 0.000,C 180.000,E1 0.000} C_DIS
LIN {X -120.652,Y 257.776,Z 50.000,A 0.000,B 0.000,C 180.000,E1 0.000} C_DIS
LIN {X -133.763,Y 251.223,Z 50.000,A 0.000,B 0.000,C 180.000,E1 0.000} C_DIS
LIN {X -146.518,Y 244.004,Z 50.000,A 0.000,B 0.000,C 180.000,E1 0.000} C_DIS
LIN {X -158.884,Y 236.139,Z 50.000,A 0.000,B 0.000,C 180.000,E1 0.000} C_DIS
LIN {X -170.829,Y 227.646,Z 50.000,A 0.000,B 0.000,C 180.000,E1 0.000} C_DIS
LIN {X -182.322,Y 218.551,Z 50.000,A 0.000,B 0.000,C 180.000,E1 0.000} C_DIS
LIN {X -193.331,Y 208.874,Z 50.000,A 0.000,B 0.000,C 180.000,E1 0.000} C_DIS
LIN {X -203.827,Y 198.645,Z 50.000,A 0.000,B 0.000,C 180.000,E1 0.000} C_DIS
LIN {X -213.783,Y 187.889,Z 50.000,A 0.000,B 0.000,C 180.000,E1 0.000} C_DIS
LIN {X -223.171,Y 176.635,Z 50.000,A 0.000,B 0.000,C 180.000,E1 0.000} C_DIS
LIN {X -231.969,Y 164.911,Z 50.000,A 0.000,B 0.000,C 180.000,E1 0.000} C_DIS
LIN {X -240.151,Y 152.752,Z 50.000,A 0.000,B 0.000,C 180.000,E1 0.000} C_DIS
LIN {X -247.696,Y 140.186,Z 50.000,A 0.000,B 0.000,C 180.000,E1 0.000} C_DIS
LIN {X -254.584,Y 127.249,Z 50.000,A 0.000,B 0.000,C 180.000,E1 0.000} C_DIS
LIN {X -260.798,Y 113.975,Z 50.000,A 0.000,B 0.000,C 180.000,E1 0.000} C_DIS
;rapid-leaky
$VEL.CP=0.3
LIN {X -246.553,Y 107.750,Z 50.000,A 0.000,B 0.000,C 180.000,E1 0.000} C_DIS
;bead-perimeter_inner
$VEL.CP=0.76
LIN {X -251.773,Y 94.916,Z 50.000,A 0.000,B 0.000,C 180.000,E1 0.000} C_DIS
LIN {X -256.324,Y 81.828,Z 50.000,A 0.000,B 0.000,C 180.000,E1 0.000} C_DIS
LIN {X -260.198,Y 68.524,Z 50.000,A 0.000,B 0.000,C 180.000,E1 0.000} C_DIS
LIN {X -263.380,Y 55.040,Z 50.000,A 0.000,B 0.000,C 180.000,E1 0.000} C_DIS
LIN {X -265.864,Y 41.407,Z 50.000,A 0.000,B 0.000,C 180.000,E1 0.000} C_DIS
LIN {X -267.643,Y 27.665,Z 50.000,A 0.000,B 0.000,C 180.000,E1 0.000} C_DIS
LIN {X -268.713,Y 13.851,Z 50.000,A 0.000,B 0.000,C 180.000,E1 0.000} C_DIS
LIN {X -269.069,Y 0.000,Z 50.000,A 0.000,B 0.000,C 180.000,E1 0.000} C_DIS
LIN {X -268.713,Y -13.851,Z 50.000,A 0.000,B 0.000,C 180.000,E1 0.000} C_DIS
LIN {X -267.643,Y -27.665,Z 50.000,A 0.000,B 0.000,C 180.000,E1 0.000} C_DIS
LIN {X -265.864,Y -41.407,Z 50.000,A 0.000,B 0.000,C 180.000,E1 0.000} C_DIS
LIN {X -263.380,Y -55.040,Z 50.000,A 0.000,B 0.000,C 180.000,E1 0.000} C_DIS
LIN {X -260.198,Y -68.524,Z 50.000,A 0.000,B 0.000,C 180.000,E1 0.000} C_DIS
LIN {X -256.324,Y -81.828,Z 50.000,A 0.000,B 0.000,C 180.000,E1 0.000} C_DIS
LIN {X -251.773,Y -94.916,Z 50.000,A 0.000,B 0.000,C 180.000,E1 0.000} C_DIS
LIN {X -246.553,Y -107.750,Z 50.000,A 0.000,B 0.000,C 180.000,E1 0.000} C_DIS
LIN {X -240.679,Y -120.299,Z 50.000,A 0.000,B 0.000,C 180.000,E1 0.000} C_DIS
LIN {X -234.167,Y -132.529,Z 50.000,A 0.000,B 0.000,C 180.000,E1 0.000} C_DIS
LIN {X -227.034,Y -144.409,Z 50.000,A 0.000,B 0.000,C 180.000,E1 0.000} C_DIS
LIN {X -219.300,Y -155.904,Z 50.000,A 0.000,B 0.000,C 180.000,E1 0.000} C_DIS
LIN {X -210.982,Y -166.987,Z 50.000,A 0.000,B 0.000,C 180.000,E1 0.000} C_DIS
LIN {X -202.106,Y -177.627,Z 50.000,A 0.000,B 0.000,C 180.000,E1 0.000} C_DIS
LIN {X -192.694,Y -187.796,Z 50.000,A 0.000,B 0.000,C 180.000,E1 0.000} C_DIS
LIN {X -182.772,Y -197.466,Z 50.000,A 0.000,B 0.000,C 180.000,E1 0.000} C_DIS
LIN {X -172.364,Y -206.614,Z 50.000,A 0.000,B 0.000,C 180.000,E1 0.000} C_DIS
LIN {X -161.499,Y -215.212,Z 50.000,A 0.000,B 0.000,C 180.000,E1 0.000} C_DIS
LIN {X -150.206,Y -223.241,Z 50.000,A 0.000,B 0.000,C 180.000,E1 0.000} C_DIS
LIN {X -138.516,Y -230.676,Z 50.000,A 0.000,B 0.000,C 180.000,E1 0.000} C_DIS
LIN {X -126.457,Y -237.501,Z 50.000,A 0.000,B 0.000,C 180.000,E1 0.000} C_DIS
LIN {X -114.062,Y -243.696,Z 50.000,A 0.000,B 0.000,C 180.000,E1 0.000} C_DIS
LIN {X -101.365,Y -249.246,Z 50.000,A 0.000,B 0.000,C 180.000,E1 0.000} C_DIS
LIN {X -88.401,Y -254.134,Z 50.000,A 0.000,B 0.000,C 180.000,E1 0.000} C_DIS
LIN {X -75.201,Y -258.347,Z 50.000,A 0.000,B 0.000,C 180.000,E1 0.000} C_DIS
LIN {X -61.802,Y -261.876,Z 50.000,A 0.000,B 0.000,C 180.000,E1 0.000} C_DIS
LIN {X -48.238,Y -264.710,Z 50.000,A 0.000,B 0.000,C 180.000,E1 0.000} C_DIS
LIN {X -34.548,Y -266.843,Z 50.000,A 0.000,B 0.000,C 180.000,E1 0.000} C_DIS
LIN {X -20.767,Y -268.267,Z 50.000,A 0.000,B 0.000,C 180.000,E1 0.000} C_DIS
LIN {X -6.928,Y -268.980,Z 50.000,A 0.000,B 0.000,C 180.000,E1 0.000} C_DIS
LIN {X 6.928,Y -268.980,Z 50.000,A 0.000,B 0.000,C 180.000,E1 0.000} C_DIS
LIN {X 20.767,Y -268.267,Z 50.000,A 0.000,B 0.000,C 180.000,E1 0.000} C_DIS
LIN {X 34.548,Y -266.843,Z 50.000,A 0.000,B 0.000,C 180.000,E1 0.000} C_DIS
LIN {X 48.238,Y -264.710,Z 50.000,A 0.000,B 0.000,C 180.000,E1 0.000} C_DIS
LIN {X 61.802,Y -261.876,Z 50.000,A 0.000,B 0.000,C 180.000,E1 0.000} C_DIS
LIN {X 75.201,Y -258.347,Z 50.000,A 0.000,B 0.000,C 180.000,E1 0.000} C_DIS
LIN {X 88.401,Y -254.134,Z 50.000,A 0.000,B 0.000,C 180.000,E1 0.000} C_DIS
LIN {X 101.367,Y -249.245,Z 50.000,A 0.000,B 0.000,C 180.000,E1 0.000} C_DIS
LIN {X 104.987,Y -247.664,Z 50.000,A 0.000,B 0.000,C 180.000,E1 0.000} C_DIS
LIN {X 114.061,Y -243.697,Z 50.000,A 0.000,B 0.000,C 180.000,E1 0.000} C_DIS
LIN {X 126.457,Y -237.501,Z 50.000,A 0.000,B 0.000,C 180.000,E1 0.000} C_DIS
LIN {X 138.516,Y -230.676,Z 50.000,A 0.000,B 0.000,C 180.000,E1 0.000} C_DIS
LIN {X 150.206,Y -223.241,Z 50.000,A 0.000,B 0.000,C 180.000,E1 0.000} C_DIS
LIN {X 161.499,Y -215.212,Z 50.000,A 0.000,B 0.000,C 180.000,E1 0.000} C_DIS
LIN {X 172.364,Y -206.614,Z 50.000,A 0.000,B 0.000,C 180.000,E1 0.000} C_DIS
LIN {X 182.772,Y -197.466,Z 50.000,A 0.000,B 0.000,C 180.000,E1 0.000} C_DIS
LIN {X 192.694,Y -187.796,Z 50.000,A 0.000,B 0.000,C 180.000,E1 0.000} C_DIS
LIN {X 202.106,Y -177.627,Z 50.000,A 0.000,B 0.000,C 180.000,E1 0.000} C_DIS
LIN {X 210.982,Y -166.987,Z 50.000,A 0.000,B 0.000,C 180.000,E1 0.000} C_DIS
LIN {X 219.300,Y -155.904,Z 50.000,A 0.000,B 0.000,C 180.000,E1 0.000} C_DIS
LIN {X 227.034,Y -144.409,Z 50.000,A 0.000,B 0.000,C 180.000,E1 0.000} C_DIS
LIN {X 234.167,Y -132.529,Z 50.000,A 0.000,B 0.000,C 180.000,E1 0.000} C_DIS
LIN {X 240.679,Y -120.299,Z 50.000,A 0.000,B 0.000,C 180.000,E1 0.000} C_DIS
LIN {X 246.553,Y -107.750,Z 50.000,A 0.000,B 0.000,C 180.000,E1 0.000} C_DIS
LIN {X 251.773,Y -94.916,Z 50.000,A 0.000,B 0.000,C 180.000,E1 0.000} C_DIS
LIN {X 256.324,Y -81.828,Z 50.000,A 0.000,B 0.000,C 180.000,E1 0.000} C_DIS
LIN {X 260.198,Y -68.524,Z 50.000,A 0.000,B 0.000,C 180.000,E1 0.000} C_DIS
LIN {X 263.380,Y -55.040,Z 50.000,A 0.000,B 0.000,C 180.000,E1 0.000} C_DIS
LIN {X 265.864,Y -41.407,Z 50.000,A 0.000,B 0.000,C 180.000,E1 0.000} C_DIS
LIN {X 267.643,Y -27.665,Z 50.000,A 0.000,B 0.000,C 180.000,E1 0.000} C_DIS
LIN {X 268.713,Y -13.851,Z 50.000,A 0.000,B 0.000,C 180.000,E1 0.000} C_DIS
LIN {X 269.069,Y 0.000,Z 50.000,A 0.000,B 0.000,C 180.000,E1 0.000} C_DIS
LIN {X 268.713,Y 13.851,Z 50.000,A 0.000,B 0.000,C 180.000,E1 0.000} C_DIS
LIN {X 267.643,Y 27.665,Z 50.000,A 0.000,B 0.000,C 180.000,E1 0.000} C_DIS
LIN {X 265.864,Y 41.407,Z 50.000,A 0.000,B 0.000,C 180.000,E1 0.000} C_DIS
LIN {X 263.380,Y 55.040,Z 50.000,A 0.000,B 0.000,C 180.000,E1 0.000} C_DIS
LIN {X 260.198,Y 68.524,Z 50.000,A 0.000,B 0.000,C 180.000,E1 0.000} C_DIS
LIN {X 256.324,Y 81.828,Z 50.000,A 0.000,B 0.000,C 180.000,E1 0.000} C_DIS
LIN {X 251.773,Y 94.916,Z 50.000,A 0.000,B 0.000,C 180.000,E1 0.000} C_DIS
LIN {X 246.553,Y 107.750,Z 50.000,A 0.000,B 0.000,C 180.000,E1 0.000} C_DIS
LIN {X 240.679,Y 120.299,Z 50.000,A 0.000,B 0.000,C 180.000,E1 0.000} C_DIS
LIN {X 234.167,Y 132.529,Z 50.000,A 0.000,B 0.000,C 180.000,E1 0.000} C_DIS
LIN {X 227.034,Y 144.409,Z 50.000,A 0.000,B 0.000,C 180.000,E1 0.000} C_DIS
LIN {X 219.300,Y 155.904,Z 50.000,A 0.000,B 0.000,C 180.000,E1 0.000} C_DIS
LIN {X 210.982,Y 166.987,Z 50.000,A 0.000,B 0.000,C 180.000,E1 0.000} C_DIS
LIN {X 202.106,Y 177.627,Z 50.000,A 0.000,B 0.000,C 180.000,E1 0.000} C_DIS
LIN {X 192.694,Y 187.796,Z 50.000,A 0.000,B 0.000,C 180.000,E1 0.000} C_DIS
LIN {X 182.772,Y 197.466,Z 50.000,A 0.000,B 0.000,C 180.000,E1 0.000} C_DIS
LIN {X 172.364,Y 206.614,Z 50.000,A 0.000,B 0.000,C 180.000,E1 0.000} C_DIS
LIN {X 161.499,Y 215.212,Z 50.000,A 0.000,B 0.000,C 180.000,E1 0.000} C_DIS
LIN {X 150.206,Y 223.241,Z 50.000,A 0.000,B 0.000,C 180.000,E1 0.000} C_DIS
LIN {X 138.516,Y 230.676,Z 50.000,A 0.000,B 0.000,C 180.000,E1 0.000} C_DIS
LIN {X 126.457,Y 237.501,Z 50.000,A 0.000,B 0.000,C 180.000,E1 0.000} C_DIS
LIN {X 114.062,Y 243.696,Z 50.000,A 0.000,B 0.000,C 180.000,E1 0.000} C_DIS
LIN {X 101.365,Y 249.246,Z 50.000,A 0.000,B 0.000,C 180.000,E1 0.000} C_DIS
LIN {X 88.401,Y 254.134,Z 50.000,A 0.000,B 0.000,C 180.000,E1 0.000} C_DIS
LIN {X 75.201,Y 258.347,Z 50.000,A 0.000,B 0.000,C 180.000,E1 0.000} C_DIS
LIN {X 61.802,Y 261.876,Z 50.000,A 0.000,B 0.000,C 180.000,E1 0.000} C_DIS
LIN {X 48.238,Y 264.710,Z 50.000,A 0.000,B 0.000,C 180.000,E1 0.000} C_DIS
LIN {X 34.548,Y 266.843,Z 50.000,A 0.000,B 0.000,C 180.000,E1 0.000} C_DIS
LIN {X 20.767,Y 268.267,Z 50.000,A 0.000,B 0.000,C 180.000,E1 0.000} C_DIS
LIN {X 6.928,Y 268.980,Z 50.000,A 0.000,B 0.000,C 180.000,E1 0.000} C_DIS
LIN {X -6.928,Y 268.980,Z 50.000,A 0.000,B 0.000,C 180.000,E1 0.000} C_DIS
LIN {X -20.767,Y 268.267,Z 50.000,A 0.000,B 0.000,C 180.000,E1 0.000} C_DIS
LIN {X -34.548,Y 266.843,Z 50.000,A 0.000,B 0.000,C 180.000,E1 0.000} C_DIS
LIN {X -48.238,Y 264.710,Z 50.000,A 0.000,B 0.000,C 180.000,E1 0.000} C_DIS
LIN {X -61.802,Y 261.876,Z 50.000,A 0.000,B 0.000,C 180.000,E1 0.000} C_DIS
LIN {X -75.201,Y 258.347,Z 50.000,A 0.000,B 0.000,C 180.000,E1 0.000} C_DIS
LIN {X -88.401,Y 254.134,Z 50.000,A 0.000,B 0.000,C 180.000,E1 0.000} C_DIS
LIN {X -101.367,Y 249.245,Z 50.000,A 0.000,B 0.000,C 180.000,E1 0.000} C_DIS
LIN {X -114.061,Y 243.697,Z 50.000,A 0.000,B 0.000,C 180.000,E1 0.000} C_DIS
LIN {X -126.457,Y 237.501,Z 50.000,A 0.000,B 0.000,C 180.000,E1 0.000} C_DIS
LIN {X -138.516,Y 230.676,Z 50.000,A 0.000,B 0.000,C 180.000,E1 0.000} C_DIS
LIN {X -150.206,Y 223.241,Z 50.000,A 0.000,B 0.000,C 180.000,E1 0.000} C_DIS
LIN {X -161.499,Y 215.212,Z 50.000,A 0.000,B 0.000,C 180.000,E1 0.000} C_DIS
LIN {X -172.364,Y 206.614,Z 50.000,A 0.000,B 0.000,C 180.000,E1 0.000} C_DIS
LIN {X -182.772,Y 197.466,Z 50.000,A 0.000,B 0.000,C 180.000,E1 0.000} C_DIS
LIN {X -192.694,Y 187.796,Z 50.000,A 0.000,B 0.000,C 180.000,E1 0.000} C_DIS
LIN {X -202.106,Y 177.627,Z 50.000,A 0.000,B 0.000,C 180.000,E1 0.000} C_DIS
LIN {X -210.982,Y 166.987,Z 50.000,A 0.000,B 0.000,C 180.000,E1 0.000} C_DIS
LIN {X -219.300,Y 155.904,Z 50.000,A 0.000,B 0.000,C 180.000,E1 0.000} C_DIS
LIN {X -227.034,Y 144.409,Z 50.000,A 0.000,B 0.000,C 180.000,E1 0.000} C_DIS
LIN {X -234.167,Y 132.529,Z 50.000,A 0.000,B 0.000,C 180.000,E1 0.000} C_DIS
LIN {X -240.679,Y 120.299,Z 50.000,A 0.000,B 0.000,C 180.000,E1 0.000} C_DIS
LIN {X -246.553,Y 107.750,Z 50.000,A 0.000,B 0.000,C 180.000,E1 0.000} C_DIS
;rapid-leaky
$VEL.CP=0.3
LIN {X -214.352,Y -131.029,Z 50.000,A 0.000,B 0.000,C 180.000,E1 0.000} C_DIS
;bead-sparse_infill
$VEL.CP=0.76
LIN {X -130.924,Y -214.457,Z 50.000,A 0.000,B 0.000,C 180.000,E1 0.000} C_DIS
LIN {X -129.370,Y -215.445,Z 50.000,A 0.000,B 0.000,C 180.000,E1 0.000} C_DIS
LIN {X -118.108,Y -221.820,Z 50.000,A 0.000,B 0.000,C 180.000,E1 0.000} C_DIS
LIN {X -106.531,Y -227.606,Z 50.000,A 0.000,B 0.000,C 180.000,E1 0.000} C_DIS
LIN {X -94.671,Y -232.789,Z 50.000,A 0.000,B 0.000,C 180.000,E1 0.000} C_DIS
LIN {X -82.564,Y -237.354,Z 50.000,A 0.000,B 0.000,C 180.000,E1 0.000} C_DIS
LIN {X -70.236,Y -241.289,Z 50.000,A 0.000,B 0.000,C 180.000,E1 0.000} C_DIS
LIN {X -57.722,Y -244.585,Z 50.000,A 0.000,B 0.000,C 180.000,E1 0.000} C_DIS
LIN {X -45.053,Y -247.232,Z 50.000,A 0.000,B 0.000,C 180.000,E1 0.000} C_DIS
LIN {X -32.267,Y -249.224,Z 50.000,A 0.000,B 0.000,C 180.000,E1 0.000} C_DIS
LIN {X -19.396,Y -250.554,Z 50.000,A 0.000,B 0.000,C 180.000,E1 0.000} C_DIS
LIN {X -6.470,Y -251.220,Z 50.000,A 0.000,B 0.000,C 180.000,E1 0.000} C_DIS
LIN {X 6.470,Y -251.220,Z 50.000,A 0.000,B 0.000,C 180.000,E1 0.000} C_DIS
LIN {X 19.396,Y -250.554,Z 50.000,A 0.000,B 0.000,C 180.000,E1 0.000} C_DIS
LIN {X 32.267,Y -249.224,Z 50.000,A 0.000,B 0.000,C 180.000,E1 0.000} C_DIS
LIN {X 45.053,Y -247.232,Z 50.000,A 0.000,B 0.000,C 180.000,E1 0.000} C_DIS
LIN {X 56.448,Y -244.851,Z 50.000,A 0.000,B 0.000,C 180.000,E1 0.000} C_DIS
LIN {X -244.810,Y 56.406,Z 50.000,A 0.000,B 0.000,C 180.000,E1 0.000} C_DIS
LIN {X -243.018,Y 63.999,Z 50.000,A 0.000,B 0.000,C 180.000,E1 0.000} C_DIS
LIN {X -239.400,Y 76.425,Z 50.000,A 0.000,B 0.000,C 180.000,E1 0.000} C_DIS
LIN {X -235.149,Y 88.649,Z 50.000,A 0.000,B 0.000,C 180.000,E1 0.000} C_DIS
LIN {X -230.274,Y 100.635,Z 50.000,A 0.000,B 0.000,C 180.000,E1 0.000} C_DIS
LIN {X -224.788,Y 112.355,Z 50.000,A 0.000,B 0.000,C 180.000,E1 0.000} C_DIS
LIN {X -218.705,Y 123.779,Z 50.000,A 0.000,B 0.000,C 180.000,E1 0.000} C_DIS
LIN {X -212.044,Y 134.874,Z 50.000,A 0.000,B 0.000,C 180.000,E1 0.000} C_DIS
LIN {X -204.820,Y 145.610,Z 50.000,A 0.000,B 0.000,C 180.000,E1 0.000} C_DIS
LIN {X -197.052,Y 155.961,Z 50.000,A 0.000,B 0.000,C 180.000,E1 0.000} C_DIS
LIN {X -192.656,Y 161.230,Z 50.000,A 0.000,B 0.000,C 180.000,E1 0.000} C_DIS
LIN {X 161.283,Y -192.708,Z 50.000,A 0.000,B 0.000,C 180.000,E1 0.000} C_DIS
LIN {X 170.704,Y -184.428,Z 50.000,A 0.000,B 0.000,C 180.000,E1 0.000} C_DIS
LIN {X 179.971,Y -175.396,Z 50.000,A 0.000,B 0.000,C 180.000,E1 0.000} C_DIS
LIN {X 188.762,Y -165.899,Z 50.000,A 0.000,B 0.000,C 180.000,E1 0.000} C_DIS
LIN {X 197.052,Y -155.961,Z 50.000,A 0.000,B 0.000,C 180.000,E1 0.000} C_DIS
LIN {X 204.820,Y -145.610,Z 50.000,A 0.000,B 0.000,C 180.000,E1 0.000} C_DIS
LIN {X 212.044,Y -134.874,Z 50.000,A 0.000,B 0.000,C 180.000,E1 0.000} C_DIS
LIN {X 218.705,Y -123.779,Z 50.000,A 0.000,B 0.000,C 180.000,E1 0.000} C_DIS
LIN {X 224.788,Y -112.355,Z 50.000,A 0.000,B 0.000,C 180.000,E1 0.000} C_DIS
LIN {X 228.971,Y -103.419,Z 50.000,A 0.000,B 0.000,C 180.000,E1 0.000} C_DIS
LIN {X -103.416,Y 228.967,Z 50.000,A 0.000,B 0.000,C 180.000,E1 0.000} C_DIS
LIN {X -94.674,Y 232.788,Z 50.000,A 0.000,B 0.000,C 180.000,E1 0.000} C_DIS
LIN {X -82.564,Y 237.354,Z 50.000,A 0.000,B 0.000,C 180.000,E1 0.000} C_DIS
LIN {X -70.236,Y 241.289,Z 50.000,A 0.000,B 0.000,C 180.000,E1 0.000} C_DIS
LIN {X -57.722,Y 244.585,Z 50.000,A 0.000,B 0.000,C 180.000,E1 0.000} C_DIS
LIN {X -45.053,Y 247.232,Z 50.000,A 0.000,B 0.000,C 180.000,E1 0.000} C_DIS
LIN {X -32.267,Y 249.224,Z 50.000,A 0.000,B 0.000,C 180.000,E1 0.000} C_DIS
LIN {X -19.396,Y 250.554,Z 50.000,A 0.000,B 0.000,C 180.000,E1 0.000} C_DIS
LIN {X -6.470,Y 251.220,Z 50.000,A 0.000,B 0.000,C 180.000,E1 0.000} C_DIS
LIN {X 6.470,Y 251.220,Z 50.000,A 0.000,B 0.000,C 180.000,E1 0.000} C_DIS
LIN {X 19.396,Y 250.554,Z 50.000,A 0.000,B 0.000,C 180.000,E1 0.000} C_DIS
LIN {X 32.267,Y 249.224,Z 50.000,A 0.000,B 0.000,C 180.000,E1 0.000} C_DIS
LIN {X 33.497,Y 249.032,Z 50.000,A 0.000,B 0.000,C 180.000,E1 0.000} C_DIS
LIN {X 248.972,Y 33.558,Z 50.000,A 0.000,B 0.000,C 180.000,E1 0.000} C_DIS
;rapid-leaky
$VEL.CP=0.3
LIN {X -276.847,Y -57.853,Z 60.000,A 0.000,B 0.000,C 180.000,E1 0.000} C_DIS
;bead-perimeter_outer
$VEL.CP=0.74
LIN {X -273.502,Y -72.027,Z 60.000,A 0.000,B 0.000,C 180.000,E1 0.000} C_DIS
LIN {X -269.430,Y -86.012,Z 60.000,A 0.000,B 0.000,C 180.000,E1 0.000} C_DIS
LIN {X -264.646,Y -99.768,Z 60.000,A 0.000,B 0.000,C 180.000,E1 0.000} C_DIS
LIN {X -259.159,Y -113.260,Z 60.000,A 0.000,B 0.000,C 180.000,E1 0.000} C_DIS
LIN {X -252.985,Y -126.450,Z 60.000,A 0.000,B 0.000,C 180.000,E1 0.000} C_DIS
LIN {X -246.140,Y -139.306,Z 60.000,A 0.000,B 0.000,C 180.000,E1 0.000} C_DIS
LIN {X -238.642,Y -151.792,Z 60.000,A 0.000,B 0.000,C 180.000,E1 0.000} C_DIS
LIN {X -230.511,Y -163.876,Z 60.000,A 0.000,B 0.000,C 180.000,E1 0.000} C_DIS
LIN {X -221.770,Y -175.525,Z 60.000,A 0.000,B 0.000,C 180.000,E1 0.000} C_DIS
LIN {X -212.441,Y -186.709,Z 60.000,A 0.000,B 0.000,C 180.000,E1 0.000} C_DIS
LIN {X -202.547,Y -197.397,Z 60.000,A 0.000,B 0.000,C 180.000,E1 0.000} C_DIS
LIN {X -192.117,Y -207.562,Z 60.000,A 0.000,B 0.000,C 180.000,E1 0.000} C_DIS
LIN {X -181.177,Y -217.178,Z 60.000,A 0.000,B 0.000,C 180.000,E1 0.000} C_DIS
LIN {X -169.757,Y -226.216,Z 60.000,A 0.000,B 0.000,C 180.000,E1 0.000} C_DIS
LIN {X -157.886,Y -234.655,Z 60.000,A 0.000,B 0.000,C 180.000,E1 0.000} C_DIS
LIN {X -145.597,Y -242.472,Z 60.000,A 0.000,B 0.000,C 180.000,E1 0.000} C_DIS
LIN {X -132.922,Y -249.645,Z 60.000,A 0.000,B 0.000,C 180.000,E1 0.000} C_DIS
LIN {X -119.894,Y -256.157,Z 60.000,A 0.000,B 0.000,C 180.000,E1 0.000} C_DIS
LIN {X -106.549,Y -261.989,Z 60.000,A 0.000,B 0.000,C 180.000,E1 0.000} C_DIS
LIN {X -92.920,Y -267.128,Z 60.000,A 0.000,B 0.000,C 180.000,E1 0.000} C_DIS
LIN {X -79.046,Y -271.557,Z 60.000,A 0.000,B 0.000,C 180.000,E1 0.000} C_DIS
LIN {X -64.962,Y -275.265,Z 60.000,A 0.000,B 0.000,C 180.000,E1 0.000} C_DIS
LIN {X -50.705,Y -278.244,Z 60.000,A 0.000,B 0.000,C 180.000,E1 0.000} C_DIS
LIN {X -36.314,Y -280.486,Z 60.000,A 0.000,B 0.000,C 180.000,E1 0.000} C_DIS
LIN {X -21.828,Y -281.983,Z 60.000,A 0.000,B 0.000,C 180.000,E1 0.000} C_DIS
LIN {X -7.282,Y -282.733,Z 60.000,A 0.000,B 0.000,C 180.000,E1 0.000} C_DIS
LIN {X 7.282,Y -282.733,Z 60.000,A 0.000,B 0.000,C 180.000,E1 0.000} C_DIS
LIN {X 21.707,Y -281.990,Z 60.000,A 0.000,B 0.000,C 180.000,E1 0.000} C_DIS
LIN {X 36.314,Y -280.486,Z 60.000,A 0.000,B 0.000,C 180.000,E1 0.000} C_DIS
LIN {X 50.705,Y -278.244,Z 60.000,A 0.000,B 0.000,C 180.000,E1 0.000} C_DIS
LIN {X 64.962,Y -275.265,Z 60.000,A 0.000,B 0.000,C 180.000,E1 0.000} C_DIS
LIN {X 79.046,Y -271.557,Z 60.000,A 0.000,B 0.000,C 180.000,E1 0.000} C_DIS
LIN {X 92.920,Y -267.128,Z 60.000,A 0.000,B 0.000,C 180.000,E1 0.000} C_DIS
LIN {X 106.549,Y -261.989,Z 60.000,A 0.000,B 0.000,C 180.000,E1 0.000} C_DIS
LIN {X 119.894,Y -256.157,Z 60.000,A 0.000,B 0.000,C 180.000,E1 0.000} C_DIS
LIN {X 132.922,Y -249.645,Z 60.000,A 0.000,B 0.000,C 180.000,E1 0.000} C_DIS
LIN {X 145.597,Y -242.472,Z 60.000,A 0.000,B 0.000,C 180.000,E1 0.000} C_DIS
LIN {X 157.886,Y -234.655,Z 60.000,A 0.000,B 0.000,C 180.000,E1 0.000} C_DIS
LIN {X 169.757,Y -226.216,Z 60.000,A 0.000,B 0.000,C 180.000,E1 0.000} C_DIS
LIN {X 181.177,Y -217.178,Z 60.000,A 0.000,B 0.000,C 180.000,E1 0.000} C_DIS
LIN {X 192.117,Y -207.562,Z 60.000,A 0.000,B 0.000,C 180.000,E1 0.000} C_DIS
LIN {X 202.547,Y -197.397,Z 60.000,A 0.000,B 0.000,C 180.000,E1 0.000} C_DIS
LIN {X 212.441,Y -186.709,Z 60.000,A 0.000,B 0.000,C 180.000,E1 0.000} C_DIS
LIN {X 221.770,Y -175.525,Z 60.000,A 0.000,B 0.000,C 180.000,E1 0.000} C_DIS
LIN {X 230.511,Y -163.876,Z 60.000,A 0.000,B 0.000,C 180.000,E1 0.000} C_DIS
LIN {X 238.642,Y -151.791,Z 60.000,A 0.000,B 0.000,C 180.000,E1 0.000} C_DIS
LIN {X 246.075,Y -139.415,Z 60.000,A 0.000,B 0.000,C 180.000,E1 0.000} C_DIS
LIN {X 252.985,Y -126.450,Z 60.000,A 0.000,B 0.000,C 180.000,E1 0.000} C_DIS
LIN {X 259.159,Y -113.260,Z 60.000,A 0.000,B 0.000,C 180.000,E1 0.000} C_DIS
LIN {X 264.646,Y -99.768,Z 60.000,A 0.000,B 0.000,C 180.000,E1 0.000} C_DIS
LIN {X 269.430,Y -86.012,Z 60.000,A 0.000,B 0.000,C 180.000,E1 0.000} C_DIS
LIN {X 273.502,Y -72.027,Z 60.000,A 0.000,B 0.000,C 180.000,E1 0.000} C_DIS
LIN {X 276.847,Y -57.853,Z 60.000,A 0.000,B 0.000,C 180.000,E1 0.000} C_DIS
LIN {X 279.458,Y -43.525,Z 60.000,A 0.000,B 0.000,C 180.000,E1 0.000} C_DIS
LIN {X 281.327,Y -29.081,Z 60.000,A 0.000,B 0.000,C 180.000,E1 0.000} C_DIS
LIN {X 282.451,Y -14.559,Z 60.000,A 0.000,B 0.000,C 180.000,E1 0.000} C_DIS
LIN {X 282.826,Y 0.000,Z 60.000,A 0.000,B 0.000,C 180.000,E1 0.000} C_DIS
LIN {X 282.451,Y 14.559,Z 60.000,A 0.000,B 0.000,C 180.000,E1 0.000} C_DIS
LIN {X 281.327,Y 29.081,Z 60.000,A 0.000,B 0.000,C 180.000,E1 0.000} C_DIS
LIN {X 279.458,Y 43.525,Z 60.000,A 0.000,B 0.000,C 180.000,E1 0.000} C_DIS
LIN {X 276.847,Y 57.853,Z 60.000,A 0.000,B 0.000,C 180.000,E1 0.000} C_DIS
LIN {X 273.502,Y 72.027,Z 60.000,A 0.000,B 0.000,C 180.000,E1 0.000} C_DIS
LIN {X 269.430,Y 86.012,Z 60.000,A 0.000,B 0.000,C 180.000,E1 0.000} C_DIS
LIN {X 264.646,Y 99.768,Z 60.000,A 0.000,B 0.000,C 180.000,E1 0.000} C_DIS
LIN {X 259.159,Y 113.260,Z 60.000,A 0.000,B 0.000,C 180.000,E1 0.000} C_DIS
LIN {X 252.985,Y 126.450,Z 60.000,A 0.000,B 0.000,C 180.000,E1 0.000} C_DIS
LIN {X 246.140,Y 139.306,Z 60.000,A 0.000,B 0.000,C 180.000,E1 0.000} C_DIS
LIN {X 238.642,Y 151.792,Z 60.000,A 0.000,B 0.000,C 180.000,E1 0.000} C_DIS
LIN {X 230.511,Y 163.876,Z 60.000,A 0.000,B 0.000,C 180.000,E1 0.000} C_DIS
LIN {X 221.770,Y 175.525,Z 60.000,A 0.000,B 0.000,C 180.000,E1 0.000} C_DIS
LIN {X 212.441,Y 186.709,Z 60.000,A 0.000,B 0.000,C 180.000,E1 0.000} C_DIS
LIN {X 202.547,Y 197.397,Z 60.000,A 0.000,B 0.000,C 180.000,E1 0.000} C_DIS
LIN {X 192.117,Y 207.562,Z 60.000,A 0.000,B 0.000,C 180.000,E1 0.000} C_DIS
LIN {X 181.177,Y 217.178,Z 60.000,A 0.000,B 0.000,C 180.000,E1 0.000} C_DIS
LIN {X 169.757,Y 226.216,Z 60.000,A 0.000,B 0.000,C 180.000,E1 0.000} C_DIS
LIN {X 157.886,Y 234.655,Z 60.000,A 0.000,B 0.000,C 180.000,E1 0.000} C_DIS
LIN {X 145.597,Y 242.472,Z 60.000,A 0.000,B 0.000,C 180.000,E1 0.000} C_DIS
LIN {X 132.922,Y 249.645,Z 60.000,A 0.000,B 0.000,C 180.000,E1 0.000} C_DIS
LIN {X 119.894,Y 256.157,Z 60.000,A 0.000,B 0.000,C 180.000,E1 0.000} C_DIS
LIN {X 106.549,Y 261.989,Z 60.000,A 0.000,B 0.000,C 180.000,E1 0.000} C_DIS
LIN {X 92.920,Y 267.128,Z 60.000,A 0.000,B 0.000,C 180.000,E1 0.000} C_DIS
LIN {X 79.046,Y 271.557,Z 60.000,A 0.000,B 0.000,C 180.000,E1 0.000} C_DIS
LIN {X 64.962,Y 275.265,Z 60.000,A 0.000,B 0.000,C 180.000,E1 0.000} C_DIS
LIN {X 50.705,Y 278.244,Z 60.000,A 0.000,B 0.000,C 180.000,E1 0.000} C_DIS
LIN {X 36.314,Y 280.486,Z 60.000,A 0.000,B 0.000,C 180.000,E1 0.000} C_DIS
LIN {X 21.828,Y 281.983,Z 60.000,A 0.000,B 0.000,C 180.000,E1 0.000} C_DIS
LIN {X 7.282,Y 282.733,Z 60.000,A 0.000,B 0.000,C 180.000,E1 0.000} C_DIS
LIN {X -7.282,Y 282.733,Z 60.000,A 0.000,B 0.000,C 180.000,E1 0.000} C_DIS
LIN {X -21.707,Y 281.990,Z 60.000,A 0.000,B 0.000,C 180.000,E1 0.000} C_DIS
LIN {X -36.314,Y 280.486,Z 60.000,A 0.000,B 0.000,C 180.000,E1 0.000} C_DIS
LIN {X -50.705,Y 278.244,Z 60.000,A 0.000,B 0.000,C 180.000,E1 0.000} C_DIS
LIN {X -64.962,Y 275.265,Z 60.000,A 0.000,B 0.000,C 180.000,E1 0.000} C_DIS
LIN {X -79.046,Y 271.557,Z 60.000,A 0.000,B 0.000,C 180.000,E1 0.000} C_DIS
LIN {X -92.920,Y 267.128,Z 60.000,A 0.000,B 0.000,C 180.000,E1 0.000} C_DIS
LIN {X -106.549,Y 261.989,Z 60.000,A 0.000,B 0.000,C 180.000,E1 0.000} C_DIS
LIN {X -119.894,Y 256.157,Z 60.000,A 0.000,B 0.000,C 180.000,E1 0.000} C_DIS
LIN {X -132.922,Y 249.645,Z 60.000,A 0.000,B 0.000,C 180.000,E1 0.000} C_DIS
LIN {X -145.597,Y 242.472,Z 60.000,A 0.000,B 0.000,C 180.000,E1 0.000} C_DIS
LIN {X -157.886,Y 234.655,Z 60.000,A 0.000,B 0.000,C 180.000,E1 0.000} C_DIS
LIN {X -169.757,Y 226.216,Z 60.000,A 0.000,B 0.000,C 180.000,E1 0.000} C_DIS
LIN {X -181.177,Y 217.178,Z 60.000,A 0.000,B 0.000,C 180.000,E1 0.000} C_DIS
LIN {X -192.117,Y 207.562,Z 60.000,A 0.000,B 0.000,C 180.000,E1 0.000} C_DIS
LIN {X -202.547,Y 197.397,Z 60.000,A 0.000,B 0.000,C 180.000,E1 0.000} C_DIS
LIN {X -212.441,Y 186.709,Z 60.000,A 0.000,B 0.000,C 180.000,E1 0.000} C_DIS
LIN {X -221.770,Y 175.525,Z 60.000,A 0.000,B 0.000,C 180.000,E1 0.000} C_DIS
LIN {X -230.511,Y 163.876,Z 60.000,A 0.000,B 0.000,C 180.000,E1 0.000} C_DIS
LIN {X -238.642,Y 151.791,Z 60.000,A 0.000,B 0.000,C 180.000,E1 0.000} C_DIS
LIN {X -246.137,Y 139.312,Z 60.000,A 0.000,B 0.000,C 180.000,E1 0.000} C_DIS
LIN {X -252.985,Y 126.450,Z 60.000,A 0.000,B 0.000,C 180.000,E1 0.000} C_DIS
LIN {X -259.159,Y 113.260,Z 60.000,A 0.000,B 0.000,C 180.000,E1 0.000} C_DIS
LIN {X -264.646,Y 99.768,Z 60.000,A 0.000,B 0.000,C 180.000,E1 0.000} C_DIS
LIN {X -269.430,Y 86.012,Z 60.000,A 0.000,B 0.000,C 180.000,E1 0.000} C_DIS
LIN {X -273.502,Y 72.027,Z 60.000,A 0.000,B 0.000,C 180.000,E1 0.000} C_DIS
LIN {X -276.847,Y 57.853,Z 60.000,A 0.000,B 0.000,C 180.000,E1 0.000} C_DIS
LIN {X -279.458,Y 43.525,Z 60.000,A 0.000,B 0.000,C 180.000,E1 0.000} C_DIS
LIN {X -281.327,Y 29.081,Z 60.000,A 0.000,B 0.000,C 180.000,E1 0.000} C_DIS
LIN {X -282.451,Y 14.559,Z 60.000,A 0.000,B 0.000,C 180.000,E1 0.000} C_DIS
LIN {X -282.826,Y 0.000,Z 60.000,A 0.000,B 0.000,C 180.000,E1 0.000} C_DIS
LIN {X -282.451,Y -14.559,Z 60.000,A 0.000,B 0.000,C 180.000,E1 0.000} C_DIS
LIN {X -281.327,Y -29.081,Z 60.000,A 0.000,B 0.000,C 180.000,E1 0.000} C_DIS
LIN {X -279.458,Y -43.525,Z 60.000,A 0.000,B 0.000,C 180.000,E1 0.000} C_DIS
LIN {X -276.847,Y -57.853,Z 60.000,A 0.000,B 0.000,C 180.000,E1 0.000} C_DIS
;rapid-leaky
$VEL.CP=0.3
LIN {X -261.631,Y -54.673,Z 60.000,A 0.000,B 0.000,C 180.000,E1 0.000} C_DIS
;bead-perimeter_inner
$VEL.CP=0.74
LIN {X -258.469,Y -68.068,Z 60.000,A 0.000,B 0.000,C 180.000,E1 0.000} C_DIS
LIN {X -254.621,Y -81.285,Z 60.000,A 0.000,B 0.000,C 180.000,E1 0.000} C_DIS
LIN {X -250.100,Y -94.284,Z 60.000,A 0.000,B 0.000,C 180.000,E1 0.000} C_DIS
LIN {X -244.915,Y -107.034,Z 60.000,A 0.000,B 0.000,C 180.000,E1 0.000} C_DIS
LIN {X -239.080,Y -119.500,Z 60.000,A 0.000,B 0.000,C 180.000,E1 0.000} C_DIS
LIN {X -232.611,Y -131.649,Z 60.000,A 0.000,B 0.000,C 180.000,E1 0.000} C_DIS
LIN {X -225.526,Y -143.448,Z 60.000,A 0.000,B 0.000,C 180.000,E1 0.000} C_DIS
LIN {X -217.841,Y -154.869,Z 60.000,A 0.000,B 0.000,C 180.000,E1 0.000} C_DIS
LIN {X -209.580,Y -165.878,Z 60.000,A 0.000,B 0.000,C 180.000,E1 0.000} C_DIS
LIN {X -200.764,Y -176.447,Z 60.000,A 0.000,B 0.000,C 180.000,E1 0.000} C_DIS
LIN {X -191.414,Y -186.548,Z 60.000,A 0.000,B 0.000,C 180.000,E1 0.000} C_DIS
LIN {X -181.558,Y -196.154,Z 60.000,A 0.000,B 0.000,C 180.000,E1 0.000} C_DIS
LIN {X -171.219,Y -205.241,Z 60.000,A 0.000,B 0.000,C 180.000,E1 0.000} C_DIS
LIN {X -160.427,Y -213.782,Z 60.000,A 0.000,B 0.000,C 180.000,E1 0.000} C_DIS
LIN {X -149.208,Y -221.757,Z 60.000,A 0.000,B 0.000,C 180.000,E1 0.000} C_DIS
LIN {X -137.594,Y -229.145,Z 60.000,A 0.000,B 0.000,C 180.000,E1 0.000} C_DIS
LIN {X -125.616,Y -235.924,Z 60.000,A 0.000,B 0.000,C 180.000,E1 0.000} C_DIS
LIN {X -113.304,Y -242.078,Z 60.000,A 0.000,B 0.000,C 180.000,E1 0.000} C_DIS
LIN {X -100.692,Y -247.590,Z 60.000,A 0.000,B 0.000,C 180.000,E1 0.000} C_DIS
LIN {X -87.813,Y -252.446,Z 60.000,A 0.000,B 0.000,C 180.000,E1 0.000} C_DIS
LIN {X -74.702,Y -256.631,Z 60.000,A 0.000,B 0.000,C 180.000,E1 0.000} C_DIS
LIN {X -61.392,Y -260.135,Z 60.000,A 0.000,B 0.000,C 180.000,E1 0.000} C_DIS
LIN {X -47.918,Y -262.951,Z 60.000,A 0.000,B 0.000,C 180.000,E1 0.000} C_DIS
LIN {X -34.318,Y -265.070,Z 60.000,A 0.000,B 0.000,C 180.000,E1 0.000} C_DIS
LIN {X -20.629,Y -266.485,Z 60.000,A 0.000,B 0.000,C 180.000,E1 0.000} C_DIS
LIN {X -6.882,Y -267.193,Z 60.000,A 0.000,B 0.000,C 180.000,E1 0.000} C_DIS
LIN {X 6.882,Y -267.193,Z 60.000,A 0.000,B 0.000,C 180.000,E1 0.000} C_DIS
LIN {X 20.628,Y -266.485,Z 60.000,A 0.000,B 0.000,C 180.000,E1 0.000} C_DIS
LIN {X 34.318,Y -265.070,Z 60.000,A 0.000,B 0.000,C 180.000,E1 0.000} C_DIS
LIN {X 47.918,Y -262.951,Z 60.000,A 0.000,B 0.000,C 180.000,E1 0.000} C_DIS
LIN {X 61.392,Y -260.135,Z 60.000,A 0.000,B 0.000,C 180.000,E1 0.000} C_DIS
LIN {X 74.702,Y -256.631,Z 60.000,A 0.000,B 0.000,C 180.000,E1 0.000} C_DIS
LIN {X 87.813,Y -252.446,Z 60.000,A 0.000,B 0.000,C 180.000,E1 0.000} C_DIS
LIN {X 100.692,Y -247.590,Z 60.000,A 0.000,B 0.000,C 180.000,E1 0.000} C_DIS
LIN {X 113.304,Y -242.078,Z 60.000,A 0.000,B 0.000,C 180.000,E1 0.000} C_DIS
LIN {X 125.616,Y -235.924,Z 60.000,A 0.000,B 0.000,C 180.000,E1 0.000} C_DIS
LIN {X 137.594,Y -229.145,Z 60.000,A 0.000,B 0.000,C 180.000,E1 0.000} C_DIS
LIN {X 149.208,Y -221.757,Z 60.000,A 0.000,B 0.000,C 180.000,E1 0.000} C_DIS
LIN {X 160.427,Y -213.782,Z 60.000,A 0.000,B 0.000,C 180.000,E1 0.000} C_DIS
LIN {X 171.219,Y -205.241,Z 60.000,A 0.000,B 0.000,C 180.000,E1 0.000} C_DIS
LIN {X 181.558,Y -196.154,Z 60.000,A 0.000,B 0.000,C 180.000,E1 0.000} C_DIS
LIN {X 191.414,Y -186.548,Z 60.000,A 0.000,B 0.000,C 180.000,E1 0.000} C_DIS
LIN {X 200.764,Y -176.447,Z 60.000,A 0.000,B 0.000,C 180.000,E1 0.000} C_DIS
LIN {X 209.580,Y -165.878,Z 60.000,A 0.000,B 0.000,C 180.000,E1 0.000} C_DIS
LIN {X 217.841,Y -154.869,Z 60.000,A 0.000,B 0.000,C 180.000,E1 0.000} C_DIS
LIN {X 225.526,Y -143.448,Z 60.000,A 0.000,B 0.000,C 180.000,E1 0.000} C_DIS
LIN {X 232.607,Y -131.657,Z 60.000,A 0.000,B 0.000,C 180.000,E1 0.000} C_DIS
LIN {X 239.080,Y -119.500,Z 60.000,A 0.000,B 0.000,C 180.000,E1 0.000} C_DIS
LIN {X 244.915,Y -107.034,Z 60.000,A 0.000,B 0.000,C 180.000,E1 0.000} C_DIS
LIN {X 250.100,Y -94.284,Z 60.000,A 0.000,B 0.000,C 180.000,E1 0.000} C_DIS
LIN {X 254.621,Y -81.285,Z 60.000,A 0.000,B 0.000,C 180.000,E1 0.000} C_DIS
LIN {X 258.469,Y -68.068,Z 60.000,A 0.000,B 0.000,C 180.000,E1 0.000} C_DIS
LIN {X 261.631,Y -54.673,Z 60.000,A 0.000,B 0.000,C 180.000,E1 0.000} C_DIS
LIN {X 264.097,Y -41.133,Z 60.000,A 0.000,B 0.000,C 180.000,E1 0.000} C_DIS
LIN {X 265.864,Y -27.482,Z 60.000,A 0.000,B 0.000,C 180.000,E1 0.000} C_DIS
LIN {X 266.927,Y -13.759,Z 60.000,A 0.000,B 0.000,C 180.000,E1 0.000} C_DIS
LIN {X 267.281,Y 0.000,Z 60.000,A 0.000,B 0.000,C 180.000,E1 0.000} C_DIS
LIN {X 266.927,Y 13.759,Z 60.000,A 0.000,B 0.000,C 180.000,E1 0.000} C_DIS
LIN {X 265.864,Y 27.482,Z 60.000,A 0.000,B 0.000,C 180.000,E1 0.000} C_DIS
LIN {X 264.097,Y 41.133,Z 60.000,A 0.000,B 0.000,C 180.000,E1 0.000} C_DIS
LIN {X 261.631,Y 54.673,Z 60.000,A 0.000,B 0.000,C 180.000,E1 0.000} C_DIS
LIN {X 258.469,Y 68.068,Z 60.000,A 0.000,B 0.000,C 180.000,E1 0.000} C_DIS
LIN {X 254.621,Y 81.285,Z 60.000,A 0.000,B 0.000,C 180.000,E1 0.000} C_DIS
LIN {X 250.100,Y 94.284,Z 60.000,A 0.000,B 0.000,C 180.000,E1 0.000} C_DIS
LIN {X 244.915,Y 107.034,Z 60.000,A 0.000,B 0.000,C 180.000,E1 0.000} C_DIS
LIN {X 239.080,Y 119.500,Z 60.000,A 0.000,B 0.000,C 180.000,E1 0.000} C_DIS
LIN {X 232.611,Y 131.649,Z 60.000,A 0.000,B 0.000,C 180.000,E1 0.000} C_DIS
LIN {X 225.526,Y 143.448,Z 60.000,A 0.000,B 0.000,C 180.000,E1 0.000} C_DIS
LIN {X 217.841,Y 154.869,Z 60.000,A 0.000,B 0.000,C 180.000,E1 0.000} C_DIS
LIN {X 209.580,Y 165.878,Z 60.000,A 0.000,B 0.000,C 180.000,E1 0.000} C_DIS
LIN {X 200.764,Y 176.447,Z 60.000,A 0.000,B 0.000,C 180.000,E1 0.000} C_DIS
LIN {X 191.414,Y 186.548,Z 60.000,A 0.000,B 0.000,C 180.000,E1 0.000} C_DIS
LIN {X 181.558,Y 196.154,Z 60.000,A 0.000,B 0.000,C 180.000,E1 0.000} C_DIS
LIN {X 171.219,Y 205.241,Z 60.000,A 0.000,B 0.000,C 180.000,E1 0.000} C_DIS
LIN {X 160.427,Y 213.782,Z 60.000,A 0.000,B 0.000,C 180.000,E1 0.000} C_DIS
LIN {X 149.208,Y 221.757,Z 60.000,A 0.000,B 0.000,C 180.000,E1 0.000} C_DIS
LIN {X 137.594,Y 229.145,Z 60.000,A 0.000,B 0.000,C 180.000,E1 0.000} C_DIS
LIN {X 125.616,Y 235.924,Z 60.000,A 0.000,B 0.000,C 180.000,E1 0.000} C_DIS
LIN {X 113.304,Y 242.078,Z 60.000,A 0.000,B 0.000,C 180.000,E1 0.000} C_DIS
LIN {X 100.692,Y 247.590,Z 60.000,A 0.000,B 0.000,C 180.000,E1 0.000} C_DIS
LIN {X 87.813,Y 252.446,Z 60.000,A 0.000,B 0.000,C 180.000,E1 0.000} C_DIS
LIN {X 74.702,Y 256.631,Z 60.000,A 0.000,B 0.000,C 180.000,E1 0.000} C_DIS
LIN {X 61.392,Y 260.135,Z 60.000,A 0.000,B 0.000,C 180.000,E1 0.000} C_DIS
LIN {X 47.918,Y 262.951,Z 60.000,A 0.000,B 0.000,C 180.000,E1 0.000} C_DIS
LIN {X 34.318,Y 265.070,Z 60.000,A 0.000,B 0.000,C 180.000,E1 0.000} C_DIS
LIN {X 20.629,Y 266.485,Z 60.000,A 0.000,B 0.000,C 180.000,E1 0.000} C_DIS
LIN {X 6.882,Y 267.193,Z 60.000,A 0.000,B 0.000,C 180.000,E1 0.000} C_DIS
LIN {X -6.882,Y 267.193,Z 60.000,A 0.000,B 0.000,C 180.000,E1 0.000} C_DIS
LIN {X -20.628,Y 266.485,Z 60.000,A 0.000,B 0.000,C 180.000,E1 0.000} C_DIS
LIN {X -34.318,Y 265.070,Z 60.000,A 0.000,B 0.000,C 180.000,E1 0.000} C_DIS
LIN {X -47.918,Y 262.951,Z 60.000,A 0.000,B 0.000,C 180.000,E1 0.000} C_DIS
LIN {X -61.392,Y 260.135,Z 60.000,A 0.000,B 0.000,C 180.000,E1 0.000} C_DIS
LIN {X -74.702,Y 256.631,Z 60.000,A 0.000,B 0.000,C 180.000,E1 0.000} C_DIS
LIN {X -87.813,Y 252.446,Z 60.000,A 0.000,B 0.000,C 180.000,E1 0.000} C_DIS
LIN {X -100.692,Y 247.590,Z 60.000,A 0.000,B 0.000,C 180.000,E1 0.000} C_DIS
LIN {X -113.304,Y 242.078,Z 60.000,A 0.000,B 0.000,C 180.000,E1 0.000} C_DIS
LIN {X -125.616,Y 235.924,Z 60.000,A 0.000,B 0.000,C 180.000,E1 0.000} C_DIS
LIN {X -137.594,Y 229.145,Z 60.000,A 0.000,B 0.000,C 180.000,E1 0.000} C_DIS
LIN {X -149.208,Y 221.757,Z 60.000,A 0.000,B 0.000,C 180.000,E1 0.000} C_DIS
LIN {X -160.427,Y 213.782,Z 60.000,A 0.000,B 0.000,C 180.000,E1 0.000} C_DIS
LIN {X -171.219,Y 205.241,Z 60.000,A 0.000,B 0.000,C 180.000,E1 0.000} C_DIS
LIN {X -181.558,Y 196.154,Z 60.000,A 0.000,B 0.000,C 180.000,E1 0.000} C_DIS
LIN {X -191.414,Y 186.548,Z 60.000,A 0.000,B 0.000,C 180.000,E1 0.000} C_DIS
LIN {X -200.764,Y 176.447,Z 60.000,A 0.000,B 0.000,C 180.000,E1 0.000} C_DIS
LIN {X -209.580,Y 165.878,Z 60.000,A 0.000,B 0.000,C 180.000,E1 0.000} C_DIS
LIN {X -217.841,Y 154.869,Z 60.000,A 0.000,B 0.000,C 180.000,E1 0.000} C_DIS
LIN {X -225.526,Y 143.448,Z 60.000,A 0.000,B 0.000,C 180.000,E1 0.000} C_DIS
LIN {X -232.607,Y 131.657,Z 60.000,A 0.000,B 0.000,C 180.000,E1 0.000} C_DIS
LIN {X -239.080,Y 119.500,Z 60.000,A 0.000,B 0.000,C 180.000,E1 0.000} C_DIS
LIN {X -244.915,Y 107.034,Z 60.000,A 0.000,B 0.000,C 180.000,E1 0.000} C_DIS
LIN {X -250.100,Y 94.284,Z 60.000,A 0.000,B 0.000,C 180.000,E1 0.000} C_DIS
LIN {X -254.621,Y 81.285,Z 60.000,A 0.000,B 0.000,C 180.000,E1 0.000} C_DIS
LIN {X -258.469,Y 68.068,Z 60.000,A 0.000,B 0.000,C 180.000,E1 0.000} C_DIS
LIN {X -261.631,Y 54.673,Z 60.000,A 0.000,B 0.000,C 180.000,E1 0.000} C_DIS
LIN {X -264.097,Y 41.133,Z 60.000,A 0.000,B 0.000,C 180.000,E1 0.000} C_DIS
LIN {X -265.864,Y 27.482,Z 60.000,A 0.000,B 0.000,C 180.000,E1 0.000} C_DIS
LIN {X -266.927,Y 13.759,Z 60.000,A 0.000,B 0.000,C 180.000,E1 0.000} C_DIS
LIN {X -267.281,Y 0.000,Z 60.000,A 0.000,B 0.000,C 180.000,E1 0.000} C_DIS
LIN {X -266.927,Y -13.759,Z 60.000,A 0.000,B 0.000,C 180.000,E1 0.000} C_DIS
LIN {X -265.864,Y -27.482,Z 60.000,A 0.000,B 0.000,C 180.000,E1 0.000} C_DIS
LIN {X -264.097,Y -41.133,Z 60.000,A 0.000,B 0.000,C 180.000,E1 0.000} C_DIS
LIN {X -261.631,Y -54.673,Z 60.000,A 0.000,B 0.000,C 180.000,E1 0.000} C_DIS
;rapid-leaky
$VEL.CP=0.3
LIN {X -208.617,Y 136.765,Z 60.000,A 0.000,B 0.000,C 180.000,E1 0.000} C_DIS
;bead-sparse_infill
$VEL.CP=0.74
LIN {X -136.745,Y 208.637,Z 60.000,A 0.000,B 0.000,C 180.000,E1 0.000} C_DIS
LIN {X -128.448,Y 213.914,Z 60.000,A 0.000,B 0.000,C 180.000,E1 0.000} C_DIS
LIN {X -117.267,Y 220.242,Z 60.000,A 0.000,B 0.000,C 180.000,E1 0.000} C_DIS
LIN {X -105.773,Y 225.988,Z 60.000,A 0.000,B 0.000,C 180.000,E1 0.000} C_DIS
LIN {X -93.999,Y 231.133,Z 60.000,A 0.000,B 0.000,C 180.000,E1 0.000} C_DIS
LIN {X -81.976,Y 235.666,Z 60.000,A 0.000,B 0.000,C 180.000,E1 0.000} C_DIS
LIN {X -69.737,Y 239.573,Z 60.000,A 0.000,B 0.000,C 180.000,E1 0.000} C_DIS
LIN {X -57.312,Y 242.845,Z 60.000,A 0.000,B 0.000,C 180.000,E1 0.000} C_DIS
LIN {X -44.733,Y 245.473,Z 60.000,A 0.000,B 0.000,C 180.000,E1 0.000} C_DIS
LIN {X -32.037,Y 247.451,Z 60.000,A 0.000,B 0.000,C 180.000,E1 0.000} C_DIS
LIN {X -19.258,Y 248.772,Z 60.000,A 0.000,B 0.000,C 180.000,E1 0.000} C_DIS
LIN {X -6.425,Y 249.433,Z 60.000,A 0.000,B 0.000,C 180.000,E1 0.000} C_DIS
LIN {X 6.425,Y 249.433,Z 60.000,A 0.000,B 0.000,C 180.000,E1 0.000} C_DIS
LIN {X 19.258,Y 248.772,Z 60.000,A 0.000,B 0.000,C 180.000,E1 0.000} C_DIS
LIN {X 32.037,Y 247.451,Z 60.000,A 0.000,B 0.000,C 180.000,E1 0.000} C_DIS
LIN {X 44.732,Y 245.473,Z 60.000,A 0.000,B 0.000,C 180.000,E1 0.000} C_DIS
LIN {X 54.937,Y 243.341,Z 60.000,A 0.000,B 0.000,C 180.000,E1 0.000} C_DIS
LIN {X -243.324,Y -54.921,Z 60.000,A 0.000,B 0.000,C 180.000,E1 0.000} C_DIS
LIN {X -241.289,Y -63.543,Z 60.000,A 0.000,B 0.000,C 180.000,E1 0.000} C_DIS
LIN {X -237.697,Y -75.882,Z 60.000,A 0.000,B 0.000,C 180.000,E1 0.000} C_DIS
LIN {X -233.476,Y -88.018,Z 60.000,A 0.000,B 0.000,C 180.000,E1 0.000} C_DIS
LIN {X -228.636,Y -99.920,Z 60.000,A 0.000,B 0.000,C 180.000,E1 0.000} C_DIS
LIN {X -223.189,Y -111.556,Z 60.000,A 0.000,B 0.000,C 180.000,E1 0.000} C_DIS
LIN {X -217.150,Y -122.898,Z 60.000,A 0.000,B 0.000,C 180.000,E1 0.000} C_DIS
LIN {X -210.535,Y -133.913,Z 60.000,A 0.000,B 0.000,C 180.000,E1 0.000} C_DIS
LIN {X -203.361,Y -144.575,Z 60.000,A 0.000,B 0.000,C 180.000,E1 0.000} C_DIS
LIN {X -195.649,Y -154.853,Z 60.000,A 0.000,B 0.000,C 180.000,E1 0.000} C_DIS
LIN {X -191.388,Y -159.962,Z 60.000,A 0.000,B 0.000,C 180.000,E1 0.000} C_DIS
LIN {X 160.016,Y 191.442,Z 60.000,A 0.000,B 0.000,C 180.000,E1 0.000} C_DIS
LIN {X 169.490,Y 183.116,Z 60.000,A 0.000,B 0.000,C 180.000,E1 0.000} C_DIS
LIN {X 178.691,Y 174.148,Z 60.000,A 0.000,B 0.000,C 180.000,E1 0.000} C_DIS
LIN {X 187.420,Y 164.718,Z 60.000,A 0.000,B 0.000,C 180.000,E1 0.000} C_DIS
LIN {X 195.649,Y 154.853,Z 60.000,A 0.000,B 0.000,C 180.000,E1 0.000} C_DIS
LIN {X 203.361,Y 144.575,Z 60.000,A 0.000,B 0.000,C 180.000,E1 0.000} C_DIS
LIN {X 210.535,Y 133.913,Z 60.000,A 0.000,B 0.000,C 180.000,E1 0.000} C_DIS
LIN {X 217.150,Y 122.898,Z 60.000,A 0.000,B 0.000,C 180.000,E1 0.000} C_DIS
LIN {X 223.189,Y 111.556,Z 60.000,A 0.000,B 0.000,C 180.000,E1 0.000} C_DIS
LIN {X 227.627,Y 102.075,Z 60.000,A 0.000,B 0.000,C 180.000,E1 0.000} C_DIS
LIN {X -102.059,Y -227.611,Z 60.000,A 0.000,B 0.000,C 180.000,E1 0.000} C_DIS
LIN {X -93.999,Y -231.133,Z 60.000,A 0.000,B 0.000,C 180.000,E1 0.000} C_DIS
LIN {X -81.975,Y -235.666,Z 60.000,A 0.000,B 0.000,C 180.000,E1 0.000} C_DIS
LIN {X -69.737,Y -239.573,Z 60.000,A 0.000,B 0.000,C 180.000,E1 0.000} C_DIS
LIN {X -57.312,Y -242.845,Z 60.000,A 0.000,B 0.000,C 180.000,E1 0.000} C_DIS
LIN {X -44.732,Y -245.473,Z 60.000,A 0.000,B 0.000,C 180.000,E1 0.000} C_DIS
LIN {X -32.037,Y -247.451,Z 60.000,A 0.000,B 0.000,C 180.000,E1 0.000} C_DIS
LIN {X -19.258,Y -248.772,Z 60.000,A 0.000,B 0.000,C 180.000,E1 0.000} C_DIS
LIN {X -6.425,Y -249.433,Z 60.000,A 0.000,B 0.000,C 180.000,E1 0.000} C_DIS
LIN {X 6.425,Y -249.433,Z 60.000,A 0.000,B 0.000,C 180.000,E1 0.000} C_DIS
LIN {X 19.258,Y -248.772,Z 60.000,A 0.000,B 0.000,C 180.000,E1 0.000} C_DIS
LIN {X 32.037,Y -247.451,Z 60.000,A 0.000,B 0.000,C 180.000,E1 0.000} C_DIS
LIN {X 35.640,Y -246.890,Z 60.000,A 0.000,B 0.000,C 180.000,E1 0.000} C_DIS
LIN {X 246.902,Y -35.627,Z 60.000,A 0.000,B 0.000,C 180.000,E1 0.000} C_DIS
;rapid-leaky
$VEL.CP=0.3
LIN {X 277.185,Y -43.170,Z 70.000,A 0.000,B 0.000,C 180.000,E1 0.000} C_DIS
;bead-perimeter_outer
$VEL.CP=0.74
LIN {X 279.040,Y -28.844,Z 70.000,A 0.000,B 0.000,C 180.000,E1 0.000} C_DIS
LIN {X 280.155,Y -14.442,Z 70.000,A 0.000,B 0.000,C 180.000,E1 0.000} C_DIS
LIN {X 280.526,Y 0.000,Z 70.000,A 0.000,B 0.000,C 180.000,E1 0.000} C_DIS
LIN {X 280.155,Y 14.442,Z 70.000,A 0.000,B 0.000,C 180.000,E1 0.000} C_DIS
LIN {X 279.040,Y 28.844,Z 70.000,A 0.000,B 0.000,C 180.000,E1 0.000} C_DIS
LIN {X 277.185,Y 43.170,Z 70.000,A 0.000,B 0.000,C 180.000,E1 0.000} C_DIS
LIN {X 274.595,Y 57.383,Z 70.000,A 0.000,B 0.000,C 180.000,E1 0.000} C_DIS
LIN {X 271.277,Y 71.441,Z 70.000,A 0.000,B 0.000,C 180.000,E1 0.000} C_DIS
LIN {X 267.239,Y 85.312,Z 70.000,A 0.000,B 0.000,C 180.000,E1 0.000} C_DIS
LIN {X 262.494,Y 98.956,Z 70.000,A 0.000,B 0.000,C 180.000,E1 0.000} C_DIS
LIN {X 257.052,Y 112.337,Z 70.000,A 0.000,B 0.000,C 180.000,E1 0.000} C_DIS
LIN {X 250.928,Y 125.422,Z 70.000,A 0.000,B 0.000,C 180.000,E1 0.000} C_DIS
LIN {X 244.139,Y 138.173,Z 70.000,A 0.000,B 0.000,C 180.000,E1 0.000} C_DIS
LIN {X 236.702,Y 150.558,Z 70.000,A 0.000,B 0.000,C 180.000,E1 0.000} C_DIS
LIN {X 228.637,Y 162.543,Z 70.000,A 0.000,B 0.000,C 180.000,E1 0.000} C_DIS
LIN {X 219.968,Y 174.097,Z 70.000,A 0.000,B 0.000,C 180.000,E1 0.000} C_DIS
LIN {X 210.713,Y 185.190,Z 70.000,A 0.000,B 0.000,C 180.000,E1 0.000} C_DIS
LIN {X 200.900,Y 195.792,Z 70.000,A 0.000,B 0.000,C 180.000,E1 0.000} C_DIS
LIN {X 190.555,Y 205.874,Z 70.000,A 0.000,B 0.000,C 180.000,E1 0.000} C_DIS
LIN {X 179.703,Y 215.411,Z 70.000,A 0.000,B 0.000,C 180.000,E1 0.000} C_DIS
LIN {X 168.375,Y 224.377,Z 70.000,A 0.000,B 0.000,C 180.000,E1 0.000} C_DIS
LIN {X 156.602,Y 232.747,Z 70.000,A 0.000,B 0.000,C 180.000,E1 0.000} C_DIS
LIN {X 144.413,Y 240.500,Z 70.000,A 0.000,B 0.000,C 180.000,E1 0.000} C_DIS
LIN {X 131.840,Y 247.615,Z 70.000,A 0.000,B 0.000,C 180.000,E1 0.000} C_DIS
LIN {X 118.920,Y 254.073,Z 70.000,A 0.000,B 0.000,C 180.000,E1 0.000} C_DIS
LIN {X 105.682,Y 259.858,Z 70.000,A 0.000,B 0.000,C 180.000,E1 0.000} C_DIS
LIN {X 92.165,Y 264.955,Z 70.000,A 0.000,B 0.000,C 180.000,E1 0.000} C_DIS
LIN {X 78.403,Y 269.348,Z 70.000,A 0.000,B 0.000,C 180.000,E1 0.000} C_DIS
LIN {X 64.433,Y 273.026,Z 70.000,A 0.000,B 0.000,C 180.000,E1 0.000} C_DIS
LIN {X 50.292,Y 275.982,Z 70.000,A 0.000,B 0.000,C 180.000,E1 0.000} C_DIS
LIN {X 36.019,Y 278.204,Z 70.000,A 0.000,B 0.000,C 180.000,E1 0.000} C_DIS
LIN {X 21.650,Y 279.690,Z 70.000,A 0.000,B 0.000,C 180.000,E1 0.000} C_DIS
LIN {X 7.223,Y 280.434,Z 70.000,A 0.000,B 0.000,C 180.000,E1 0.000} C_DIS
LIN {X -7.223,Y 280.434,Z 70.000,A 0.000,B 0.000,C 180.000,E1 0.000} C_DIS
LIN {X -21.650,Y 279.690,Z 70.000,A 0.000,B 0.000,C 180.000,E1 0.000} C_DIS
LIN {X -36.019,Y 278.204,Z 70.000,A 0.000,B 0.000,C 180.000,E1 0.000} C_DIS
LIN {X -50.292,Y 275.982,Z 70.000,A 0.000,B 0.000,C 180.000,E1 0.000} C_DIS
LIN {X -64.433,Y 273.026,Z 70.000,A 0.000,B 0.000,C 180.000,E1 0.000} C_DIS
LIN {X -78.403,Y 269.348,Z 70.000,A 0.000,B 0.000,C 180.000,E1 0.000} C_DIS
LIN {X -92.165,Y 264.955,Z 70.000,A 0.000,B 0.000,C 180.000,E1 0.000} C_DIS
LIN {X -105.682,Y 259.858,Z 70.000,A 0.000,B 0.000,C 180.000,E1 0.000} C_DIS
LIN {X -118.920,Y 254.073,Z 70.000,A 0.000,B 0.000,C 180.000,E1 0.000} C_DIS
LIN {X -131.840,Y 247.615,Z 70.000,A 0.000,B 0.000,C 180.000,E1 0.000} C_DIS
LIN {X -144.413,Y 240.500,Z 70.000,A 0.000,B 0.000,C 180.000,E1 0.000} C_DIS
LIN {X -156.602,Y 232.747,Z 70.000,A 0.000,B 0.000,C 180.000,E1 0.000} C_DIS
LIN {X -168.375,Y 224.377,Z 70.000,A 0.000,B 0.000,C 180.000,E1 0.000} C_DIS
LIN {X -179.703,Y 215.411,Z 70.000,A 0.000,B 0.000,C 180.000,E1 0.000} C_DIS
LIN {X -190.555,Y 205.874,Z 70.000,A 0.000,B 0.000,C 180.000,E1 0.000} C_DIS
LIN {X -200.900,Y 195.792,Z 70.000,A 0.000,B 0.000,C 180.000,E1 0.000} C_DIS
LIN {X -210.713,Y 185.190,Z 70.000,A 0.000,B 0.000,C 180.000,E1 0.000} C_DIS
LIN {X -219.967,Y 174.097,Z 70.000,A 0.000,B 0.000,C 180.000,E1 0.000} C_DIS
LIN {X -228.637,Y 162.543,Z 70.000,A 0.000,B 0.000,C 180.000,E1 0.000} C_DIS
LIN {X -236.702,Y 150.558,Z 70.000,A 0.000,B 0.000,C 180.000,E1 0.000} C_DIS
LIN {X -244.139,Y 138.173,Z 70.000,A 0.000,B 0.000,C 180.000,E1 0.000} C_DIS
LIN {X -250.928,Y 125.422,Z 70.000,A 0.000,B 0.000,C 180.000,E1 0.000} C_DIS
LIN {X -257.052,Y 112.337,Z 70.000,A 0.000,B 0.000,C 180.000,E1 0.000} C_DIS
LIN {X -262.494,Y 98.956,Z 70.000,A 0.000,B 0.000,C 180.000,E1 0.000} C_DIS
LIN {X -267.239,Y 85.312,Z 70.000,A 0.000,B 0.000,C 180.000,E1 0.000} C_DIS
LIN {X -271.277,Y 71.441,Z 70.000,A 0.000,B 0.000,C 180.000,E1 0.000} C_DIS
LIN {X -274.595,Y 57.383,Z 70.000,A 0.000,B 0.000,C 180.000,E1 0.000} C_DIS
LIN {X -277.185,Y 43.170,Z 70.000,A 0.000,B 0.000,C 180.000,E1 0.000} C_DIS
LIN {X -279.040,Y 28.844,Z 70.000,A 0.000,B 0.000,C 180.000,E1 0.000} C_DIS
LIN {X -280.155,Y 14.442,Z 70.000,A 0.000,B 0.000,C 180.000,E1 0.000} C_DIS
LIN {X -280.526,Y 0.000,Z 70.000,A 0.000,B 0.000,C 180.000,E1 0.000} C_DIS
LIN {X -280.155,Y -14.442,Z 70.000,A 0.000,B 0.000,C 180.000,E1 0.000} C_DIS
LIN {X -279.040,Y -28.844,Z 70.000,A 0.000,B 0.000,C 180.000,E1 0.000} C_DIS
LIN {X -277.185,Y -43.170,Z 70.000,A 0.000,B 0.000,C 180.000,E1 0.000} C_DIS
LIN {X -274.595,Y -57.383,Z 70.000,A 0.000,B 0.000,C 180.000,E1 0.000} C_DIS
LIN {X -271.277,Y -71.441,Z 70.000,A 0.000,B 0.000,C 180.000,E1 0.000} C_DIS
LIN {X -267.239,Y -85.312,Z 70.000,A 0.000,B 0.000,C 180.000,E1 0.000} C_DIS
LIN {X -262.494,Y -98.956,Z 70.000,A 0.000,B 0.000,C 180.000,E1 0.000} C_DIS
LIN {X -257.052,Y -112.337,Z 70.000,A 0.000,B 0.000,C 180.000,E1 0.000} C_DIS
LIN {X -250.928,Y -125.422,Z 70.000,A 0.000,B 0.000,C 180.000,E1 0.000} C_DIS
LIN {X -244.139,Y -138.173,Z 70.000,A 0.000,B 0.000,C 180.000,E1 0.000} C_DIS
LIN {X -236.702,Y -150.558,Z 70.000,A 0.000,B 0.000,C 180.000,E1 0.000} C_DIS
LIN {X -228.637,Y -162.543,Z 70.000,A 0.000,B 0.000,C 180.000,E1 0.000} C_DIS
LIN {X -222.987,Y -170.074,Z 70.000,A 0.000,B 0.000,C 180.000,E1 0.000} C_DIS
LIN {X -219.968,Y -174.097,Z 70.000,A 0.000,B 0.000,C 180.000,E1 0.000} C_DIS
LIN {X -210.713,Y -185.190,Z 70.000,A 0.000,B 0.000,C 180.000,E1 0.000} C_DIS
LIN {X -200.900,Y -195.792,Z 70.000,A 0.000,B 0.000,C 180.000,E1 0.000} C_DIS
LIN {X -190.555,Y -205.874,Z 70.000,A 0.000,B 0.000,C 180.000,E1 0.000} C_DIS
LIN {X -179.703,Y -215.411,Z 70.000,A 0.000,B 0.000,C 180.000,E1 0.000} C_DIS
LIN {X -168.375,Y -224.377,Z 70.000,A 0.000,B 0.000,C 180.000,E1 0.000} C_DIS
LIN {X -156.602,Y -232.747,Z 70.000,A 0.000,B 0.000,C 180.000,E1 0.000} C_DIS
LIN {X -144.413,Y -240.500,Z 70.000,A 0.000,B 0.000,C 180.000,E1 0.000} C_DIS
LIN {X -131.840,Y -247.615,Z 70.000,A 0.000,B 0.000,C 180.000,E1 0.000} C_DIS
LIN {X -118.920,Y -254.073,Z 70.000,A 0.000,B 0.000,C 180.000,E1 0.000} C_DIS
LIN {X -105.682,Y -259.858,Z 70.000,A 0.000,B 0.000,C 180.000,E1 0.000} C_DIS
LIN {X -92.165,Y -264.955,Z 70.000,A 0.000,B 0.000,C 180.000,E1 0.000} C_DIS
LIN {X -78.403,Y -269.348,Z 70.000,A 0.000,B 0.000,C 180.000,E1 0.000} C_DIS
LIN {X -64.433,Y -273.026,Z 70.000,A 0.000,B 0.000,C 180.000,E1 0.000} C_DIS
LIN {X -50.292,Y -275.982,Z 70.000,A 0.000,B 0.000,C 180.000,E1 0.000} C_DIS
LIN {X -36.019,Y -278.204,Z 70.000,A 0.000,B 0.000,C 180.000,E1 0.000} C_DIS
LIN {X -21.650,Y -279.690,Z 70.000,A 0.000,B 0.000,C 180.000,E1 0.000} C_DIS
LIN {X -7.223,Y -280.434,Z 70.000,A 0.000,B 0.000,C 180.000,E1 0.000} C_DIS
LIN {X 7.223,Y -280.434,Z 70.000,A 0.000,B 0.000,C 180.000,E1 0.000} C_DIS
LIN {X 21.650,Y -279.690,Z 70.000,A 0.000,B 0.000,C 180.000,E1 0.000} C_DIS
LIN {X 36.019,Y -278.204,Z 70.000,A 0.000,B 0.000,C 180.000,E1 0.000} C_DIS
LIN {X 50.292,Y -275.982,Z 70.000,A 0.000,B 0.000,C 180.000,E1 0.000} C_DIS
LIN {X 64.433,Y -273.026,Z 70.000,A 0.000,B 0.000,C 180.000,E1 0.000} C_DIS
LIN {X 78.403,Y -269.348,Z 70.000,A 0.000,B 0.000,C 180.000,E1 0.000} C_DIS
LIN {X 92.165,Y -264.955,Z 70.000,A 0.000,B 0.000,C 180.000,E1 0.000} C_DIS
LIN {X 105.682,Y -259.858,Z 70.000,A 0.000,B 0.000,C 180.000,E1 0.000} C_DIS
LIN {X 118.920,Y -254.073,Z 70.000,A 0.000,B 0.000,C 180.000,E1 0.000} C_DIS
LIN {X 131.840,Y -247.615,Z 70.000,A 0.000,B 0.000,C 180.000,E1 0.000} C_DIS
LIN {X 144.413,Y -240.500,Z 70.000,A 0.000,B 0.000,C 180.000,E1 0.000} C_DIS
LIN {X 156.602,Y -232.747,Z 70.000,A 0.000,B 0.000,C 180.000,E1 0.000} C_DIS
LIN {X 168.375,Y -224.377,Z 70.000,A 0.000,B 0.000,C 180.000,E1 0.000} C_DIS
LIN {X 179.703,Y -215.411,Z 70.000,A 0.000,B 0.000,C 180.000,E1 0.000} C_DIS
LIN {X 190.555,Y -205.874,Z 70.000,A 0.000,B 0.000,C 180.000,E1 0.000} C_DIS
LIN {X 200.900,Y -195.792,Z 70.000,A 0.000,B 0.000,C 180.000,E1 0.000} C_DIS
LIN {X 210.713,Y -185.190,Z 70.000,A 0.000,B 0.000,C 180.000,E1 0.000} C_DIS
LIN {X 219.967,Y -174.097,Z 70.000,A 0.000,B 0.000,C 180.000,E1 0.000} C_DIS
LIN {X 228.637,Y -162.543,Z 70.000,A 0.000,B 0.000,C 180.000,E1 0.000} C_DIS
LIN {X 236.702,Y -150.558,Z 70.000,A 0.000,B 0.000,C 180.000,E1 0.000} C_DIS
LIN {X 244.139,Y -138.173,Z 70.000,A 0.000,B 0.000,C 180.000,E1 0.000} C_DIS
LIN {X 250.928,Y -125.422,Z 70.000,A 0.000,B 0.000,C 180.000,E1 0.000} C_DIS
LIN {X 257.052,Y -112.337,Z 70.000,A 0.000,B 0.000,C 180.000,E1 0.000} C_DIS
LIN {X 262.494,Y -98.956,Z 70.000,A 0.000,B 0.000,C 180.000,E1 0.000} C_DIS
LIN {X 267.239,Y -85.312,Z 70.000,A 0.000,B 0.000,C 180.000,E1 0.000} C_DIS
LIN {X 271.277,Y -71.441,Z 70.000,A 0.000,B 0.000,C 180.000,E1 0.000} C_DIS
LIN {X 274.595,Y -57.383,Z 70.000,A 0.000,B 0.000,C 180.000,E1 0.000} C_DIS
LIN {X 277.185,Y -43.170,Z 70.000,A 0.000,B 0.000,C 180.000,E1 0.000} C_DIS
;rapid-leaky
$VEL.CP=0.3
LIN {X 261.825,Y -40.778,Z 70.000,A 0.000,B 0.000,C 180.000,E1 0.000} C_DIS
;bead-perimeter_inner
$VEL.CP=0.74
LIN {X 263.577,Y -27.245,Z 70.000,A 0.000,B 0.000,C 180.000,E1 0.000} C_DIS
LIN {X 264.630,Y -13.642,Z 70.000,A 0.000,B 0.000,C 180.000,E1 0.000} C_DIS
LIN {X 264.981,Y 0.000,Z 70.000,A 0.000,B 0.000,C 180.000,E1 0.000} C_DIS
LIN {X 264.630,Y 13.642,Z 70.000,A 0.000,B 0.000,C 180.000,E1 0.000} C_DIS
LIN {X 263.577,Y 27.245,Z 70.000,A 0.000,B 0.000,C 180.000,E1 0.000} C_DIS
LIN {X 261.825,Y 40.778,Z 70.000,A 0.000,B 0.000,C 180.000,E1 0.000} C_DIS
LIN {X 259.379,Y 54.203,Z 70.000,A 0.000,B 0.000,C 180.000,E1 0.000} C_DIS
LIN {X 256.245,Y 67.482,Z 70.000,A 0.000,B 0.000,C 180.000,E1 0.000} C_DIS
LIN {X 252.430,Y 80.585,Z 70.000,A 0.000,B 0.000,C 180.000,E1 0.000} C_DIS
LIN {X 247.948,Y 93.473,Z 70.000,A 0.000,B 0.000,C 180.000,E1 0.000} C_DIS
LIN {X 242.807,Y 106.112,Z 70.000,A 0.000,B 0.000,C 180.000,E1 0.000} C_DIS
LIN {X 237.023,Y 118.472,Z 70.000,A 0.000,B 0.000,C 180.000,E1 0.000} C_DIS
LIN {X 230.610,Y 130.516,Z 70.000,A 0.000,B 0.000,C 180.000,E1 0.000} C_DIS
LIN {X 223.585,Y 142.214,Z 70.000,A 0.000,B 0.000,C 180.000,E1 0.000} C_DIS
LIN {X 215.967,Y 153.536,Z 70.000,A 0.000,B 0.000,C 180.000,E1 0.000} C_DIS
LIN {X 207.779,Y 164.449,Z 70.000,A 0.000,B 0.000,C 180.000,E1 0.000} C_DIS
LIN {X 199.036,Y 174.928,Z 70.000,A 0.000,B 0.000,C 180.000,E1 0.000} C_DIS
LIN {X 189.767,Y 184.943,Z 70.000,A 0.000,B 0.000,C 180.000,E1 0.000} C_DIS
LIN {X 179.996,Y 194.465,Z 70.000,A 0.000,B 0.000,C 180.000,E1 0.000} C_DIS
LIN {X 169.745,Y 203.474,Z 70.000,A 0.000,B 0.000,C 180.000,E1 0.000} C_DIS
LIN {X 159.045,Y 211.943,Z 70.000,A 0.000,B 0.000,C 180.000,E1 0.000} C_DIS
LIN {X 147.925,Y 219.849,Z 70.000,A 0.000,B 0.000,C 180.000,E1 0.000} C_DIS
LIN {X 136.411,Y 227.172,Z 70.000,A 0.000,B 0.000,C 180.000,E1 0.000} C_DIS
LIN {X 124.535,Y 233.894,Z 70.000,A 0.000,B 0.000,C 180.000,E1 0.000} C_DIS
LIN {X 112.330,Y 239.994,Z 70.000,A 0.000,B 0.000,C 180.000,E1 0.000} C_DIS
LIN {X 99.825,Y 245.459,Z 70.000,A 0.000,B 0.000,C 180.000,E1 0.000} C_DIS
LIN {X 87.058,Y 250.273,Z 70.000,A 0.000,B 0.000,C 180.000,E1 0.000} C_DIS
LIN {X 74.059,Y 254.422,Z 70.000,A 0.000,B 0.000,C 180.000,E1 0.000} C_DIS
LIN {X 60.863,Y 257.897,Z 70.000,A 0.000,B 0.000,C 180.000,E1 0.000} C_DIS
LIN {X 47.505,Y 260.689,Z 70.000,A 0.000,B 0.000,C 180.000,E1 0.000} C_DIS
LIN {X 34.023,Y 262.788,Z 70.000,A 0.000,B 0.000,C 180.000,E1 0.000} C_DIS
LIN {X 20.450,Y 264.192,Z 70.000,A 0.000,B 0.000,C 180.000,E1 0.000} C_DIS
LIN {X 6.823,Y 264.894,Z 70.000,A 0.000,B 0.000,C 180.000,E1 0.000} C_DIS
LIN {X -6.823,Y 264.894,Z 70.000,A 0.000,B 0.000,C 180.000,E1 0.000} C_DIS
LIN {X -20.450,Y 264.192,Z 70.000,A 0.000,B 0.000,C 180.000,E1 0.000} C_DIS
LIN {X -34.023,Y 262.788,Z 70.000,A 0.000,B 0.000,C 180.000,E1 0.000} C_DIS
LIN {X -47.505,Y 260.689,Z 70.000,A 0.000,B 0.000,C 180.000,E1 0.000} C_DIS
LIN {X -60.863,Y 257.897,Z 70.000,A 0.000,B 0.000,C 180.000,E1 0.000} C_DIS
LIN {X -74.059,Y 254.422,Z 70.000,A 0.000,B 0.000,C 180.000,E1 0.000} C_DIS
LIN {X -87.058,Y 250.273,Z 70.000,A 0.000,B 0.000,C 180.000,E1 0.000} C_DIS
LIN {X -99.825,Y 245.459,Z 70.000,A 0.000,B 0.000,C 180.000,E1 0.000} C_DIS
LIN {X -112.330,Y 239.994,Z 70.000,A 0.000,B 0.000,C 180.000,E1 0.000} C_DIS
LIN {X -124.534,Y 233.894,Z 70.000,A 0.000,B 0.000,C 180.000,E1 0.000} C_DIS
LIN {X -136.411,Y 227.172,Z 70.000,A 0.000,B 0.000,C 180.000,E1 0.000} C_DIS
LIN {X -147.925,Y 219.849,Z 70.000,A 0.000,B 0.000,C 180.000,E1 0.000} C_DIS
LIN {X -159.045,Y 211.943,Z 70.000,A 0.000,B 0.000,C 180.000,E1 0.000} C_DIS
LIN {X -169.745,Y 203.474,Z 70.000,A 0.000,B 0.000,C 180.000,E1 0.000} C_DIS
LIN {X -179.996,Y 194.465,Z 70.000,A 0.000,B 0.000,C 180.000,E1 0.000} C_DIS
LIN {X -189.767,Y 184.943,Z 70.000,A 0.000,B 0.000,C 180.000,E1 0.000} C_DIS
LIN {X -199.036,Y 174.928,Z 70.000,A 0.000,B 0.000,C 180.000,E1 0.000} C_DIS
LIN {X -207.778,Y 164.449,Z 70.000,A 0.000,B 0.000,C 180.000,E1 0.000} C_DIS
LIN {X -215.968,Y 153.536,Z 70.000,A 0.000,B 0.000,C 180.000,E1 0.000} C_DIS
LIN {X -223.585,Y 142.215,Z 70.000,A 0.000,B 0.000,C 180.000,E1 0.000} C_DIS
LIN {X -230.610,Y 130.516,Z 70.000,A 0.000,B 0.000,C 180.000,E1 0.000} C_DIS
LIN {X -237.023,Y 118.472,Z 70.000,A 0.000,B 0.000,C 180.000,E1 0.000} C_DIS
LIN {X -242.807,Y 106.112,Z 70.000,A 0.000,B 0.000,C 180.000,E1 0.000} C_DIS
LIN {X -247.948,Y 93.473,Z 70.000,A 0.000,B 0.000,C 180.000,E1 0.000} C_DIS
LIN {X -252.430,Y 80.585,Z 70.000,A 0.000,B 0.000,C 180.000,E1 0.000} C_DIS
LIN {X -256.245,Y 67.482,Z 70.000,A 0.000,B 0.000,C 180.000,E1 0.000} C_DIS
LIN {X -259.379,Y 54.203,Z 70.000,A 0.000,B 0.000,C 180.000,E1 0.000} C_DIS
LIN {X -261.825,Y 40.778,Z 70.000,A 0.000,B 0.000,C 180.000,E1 0.000} C_DIS
LIN {X -263.577,Y 27.245,Z 70.000,A 0.000,B 0.000,C 180.000,E1 0.000} C_DIS
LIN {X -264.630,Y 13.642,Z 70.000,A 0.000,B 0.000,C 180.000,E1 0.000} C_DIS
LIN {X -264.981,Y 0.000,Z 70.000,A 0.000,B 0.000,C 180.000,E1 0.000} C_DIS
LIN {X -264.630,Y -13.642,Z 70.000,A 0.000,B 0.000,C 180.000,E1 0.000} C_DIS
LIN {X -263.577,Y -27.245,Z 70.000,A 0.000,B 0.000,C 180.000,E1 0.000} C_DIS
LIN {X -261.825,Y -40.778,Z 70.000,A 0.000,B 0.000,C 180.000,E1 0.000} C_DIS
LIN {X -259.379,Y -54.203,Z 70.000,A 0.000,B 0.000,C 180.000,E1 0.000} C_DIS
LIN {X -256.245,Y -67.482,Z 70.000,A 0.000,B 0.000,C 180.000,E1 0.000} C_DIS
LIN {X -252.430,Y -80.585,Z 70.000,A 0.000,B 0.000,C 180.000,E1 0.000} C_DIS
LIN {X -247.948,Y -93.473,Z 70.000,A 0.000,B 0.000,C 180.000,E1 0.000} C_DIS
LIN {X -242.807,Y -106.112,Z 70.000,A 0.000,B 0.000,C 180.000,E1 0.000} C_DIS
LIN {X -237.023,Y -118.472,Z 70.000,A 0.000,B 0.000,C 180.000,E1 0.000} C_DIS
LIN {X -230.610,Y -130.516,Z 70.000,A 0.000,B 0.000,C 180.000,E1 0.000} C_DIS
LIN {X -223.585,Y -142.214,Z 70.000,A 0.000,B 0.000,C 180.000,E1 0.000} C_DIS
LIN {X -215.967,Y -153.536,Z 70.000,A 0.000,B 0.000,C 180.000,E1 0.000} C_DIS
LIN {X -210.557,Y -160.747,Z 70.000,A 0.000,B 0.000,C 180.000,E1 0.000} C_DIS
LIN {X -207.779,Y -164.449,Z 70.000,A 0.000,B 0.000,C 180.000,E1 0.000} C_DIS
LIN {X -199.036,Y -174.928,Z 70.000,A 0.000,B 0.000,C 180.000,E1 0.000} C_DIS
LIN {X -189.767,Y -184.943,Z 70.000,A 0.000,B 0.000,C 180.000,E1 0.000} C_DIS
LIN {X -179.996,Y -194.465,Z 70.000,A 0.000,B 0.000,C 180.000,E1 0.000} C_DIS
LIN {X -169.745,Y -203.474,Z 70.000,A 0.000,B 0.000,C 180.000,E1 0.000} C_DIS
LIN {X -159.045,Y -211.943,Z 70.000,A 0.000,B 0.000,C 180.000,E1 0.000} C_DIS
LIN {X -147.925,Y -219.849,Z 70.000,A 0.000,B 0.000,C 180.000,E1 0.000} C_DIS
LIN {X -136.411,Y -227.172,Z 70.000,A 0.000,B 0.000,C 180.000,E1 0.000} C_DIS
LIN {X -124.535,Y -233.894,Z 70.000,A 0.000,B 0.000,C 180.000,E1 0.000} C_DIS
LIN {X -112.330,Y -239.994,Z 70.000,A 0.000,B 0.000,C 180.000,E1 0.000} C_DIS
LIN {X -99.825,Y -245.459,Z 70.000,A 0.000,B 0.000,C 180.000,E1 0.000} C_DIS
LIN {X -87.058,Y -250.273,Z 70.000,A 0.000,B 0.000,C 180.000,E1 0.000} C_DIS
LIN {X -74.059,Y -254.422,Z 70.000,A 0.000,B 0.000,C 180.000,E1 0.000} C_DIS
LIN {X -60.863,Y -257.897,Z 70.000,A 0.000,B 0.000,C 180.000,E1 0.000} C_DIS
LIN {X -47.505,Y -260.689,Z 70.000,A 0.000,B 0.000,C 180.000,E1 0.000} C_DIS
LIN {X -34.023,Y -262.788,Z 70.000,A 0.000,B 0.000,C 180.000,E1 0.000} C_DIS
LIN {X -20.450,Y -264.192,Z 70.000,A 0.000,B 0.000,C 180.000,E1 0.000} C_DIS
LIN {X -6.823,Y -264.894,Z 70.000,A 0.000,B 0.000,C 180.000,E1 0.000} C_DIS
LIN {X 6.823,Y -264.894,Z 70.000,A 0.000,B 0.000,C 180.000,E1 0.000} C_DIS
LIN {X 20.450,Y -264.192,Z 70.000,A 0.000,B 0.000,C 180.000,E1 0.000} C_DIS
LIN {X 34.023,Y -262.788,Z 70.000,A 0.000,B 0.000,C 180.000,E1 0.000} C_DIS
LIN {X 47.505,Y -260.689,Z 70.000,A 0.000,B 0.000,C 180.000,E1 0.000} C_DIS
LIN {X 60.863,Y -257.897,Z 70.000,A 0.000,B 0.000,C 180.000,E1 0.000} C_DIS
LIN {X 74.059,Y -254.422,Z 70.000,A 0.000,B 0.000,C 180.000,E1 0.000} C_DIS
LIN {X 87.058,Y -250.273,Z 70.000,A 0.000,B 0.000,C 180.000,E1 0.000} C_DIS
LIN {X 99.825,Y -245.459,Z 70.000,A 0.000,B 0.000,C 180.000,E1 0.000} C_DIS
LIN {X 112.330,Y -239.994,Z 70.000,A 0.000,B 0.000,C 180.000,E1 0.000} C_DIS
LIN {X 124.534,Y -233.894,Z 70.000,A 0.000,B 0.000,C 180.000,E1 0.000} C_DIS
LIN {X 136.411,Y -227.172,Z 70.000,A 0.000,B 0.000,C 180.000,E1 0.000} C_DIS
LIN {X 147.925,Y -219.849,Z 70.000,A 0.000,B 0.000,C 180.000,E1 0.000} C_DIS
LIN {X 159.045,Y -211.943,Z 70.000,A 0.000,B 0.000,C 180.000,E1 0.000} C_DIS
LIN {X 169.745,Y -203.474,Z 70.000,A 0.000,B 0.000,C 180.000,E1 0.000} C_DIS
LIN {X 179.996,Y -194.465,Z 70.000,A 0.000,B 0.000,C 180.000,E1 0.000} C_DIS
LIN {X 189.767,Y -184.943,Z 70.000,A 0.000,B 0.000,C 180.000,E1 0.000} C_DIS
LIN {X 199.036,Y -174.928,Z 70.000,A 0.000,B 0.000,C 180.000,E1 0.000} C_DIS
LIN {X 207.778,Y -164.449,Z 70.000,A 0.000,B 0.000,C 180.000,E1 0.000} C_DIS
LIN {X 215.968,Y -153.536,Z 70.000,A 0.000,B 0.000,C 180.000,E1 0.000} C_DIS
LIN {X 223.585,Y -142.215,Z 70.000,A 0.000,B 0.000,C 180.000,E1 0.000} C_DIS
LIN {X 230.610,Y -130.516,Z 70.000,A 0.000,B 0.000,C 180.000,E1 0.000} C_DIS
LIN {X 237.023,Y -118.472,Z 70.000,A 0.000,B 0.000,C 180.000,E1 0.000} C_DIS
LIN {X 242.807,Y -106.112,Z 70.000,A 0.000,B 0.000,C 180.000,E1 0.000} C_DIS
LIN {X 247.948,Y -93.473,Z 70.000,A 0.000,B 0.000,C 180.000,E1 0.000} C_DIS
LIN {X 252.430,Y -80.585,Z 70.000,A 0.000,B 0.000,C 180.000,E1 0.000} C_DIS
LIN {X 256.245,Y -67.482,Z 70.000,A 0.000,B 0.000,C 180.000,E1 0.000} C_DIS
LIN {X 259.379,Y -54.203,Z 70.000,A 0.000,B 0.000,C 180.000,E1 0.000} C_DIS
LIN {X 261.825,Y -40.778,Z 70.000,A 0.000,B 0.000,C 180.000,E1 0.000} C_DIS
;rapid-leaky
$VEL.CP=0.3
LIN {X 38.396,Y 244.133,Z 70.000,A 0.000,B 0.000,C 180.000,E1 0.000} C_DIS
;bead-sparse_infill
$VEL.CP=0.74
LIN {X 244.222,Y 38.307,Z 70.000,A 0.000,B 0.000,C 180.000,E1 0.000} C_DIS
LIN {X 244.270,Y 38.044,Z 70.000,A 0.000,B 0.000,C 180.000,E1 0.000} C_DIS
LIN {X 245.906,Y 25.418,Z 70.000,A 0.000,B 0.000,C 180.000,E1 0.000} C_DIS
LIN {X 246.888,Y 12.728,Z 70.000,A 0.000,B 0.000,C 180.000,E1 0.000} C_DIS
LIN {X 247.215,Y 0.000,Z 70.000,A 0.000,B 0.000,C 180.000,E1 0.000} C_DIS
LIN {X 246.888,Y -12.728,Z 70.000,A 0.000,B 0.000,C 180.000,E1 0.000} C_DIS
LIN {X 245.906,Y -25.418,Z 70.000,A 0.000,B 0.000,C 180.000,E1 0.000} C_DIS
LIN {X 244.270,Y -38.044,Z 70.000,A 0.000,B 0.000,C 180.000,E1 0.000} C_DIS
LIN {X 241.988,Y -50.570,Z 70.000,A 0.000,B 0.000,C 180.000,E1 0.000} C_DIS
LIN {X 239.065,Y -62.957,Z 70.000,A 0.000,B 0.000,C 180.000,E1 0.000} C_DIS
LIN {X 235.506,Y -75.182,Z 70.000,A 0.000,B 0.000,C 180.000,E1 0.000} C_DIS
LIN {X 231.324,Y -87.206,Z 70.000,A 0.000,B 0.000,C 180.000,E1 0.000} C_DIS
LIN {X 226.528,Y -98.998,Z 70.000,A 0.000,B 0.000,C 180.000,E1 0.000} C_DIS
LIN {X 225.897,Y -100.345,Z 70.000,A 0.000,B 0.000,C 180.000,E1 0.000} C_DIS
LIN {X -100.312,Y 225.864,Z 70.000,A 0.000,B 0.000,C 180.000,E1 0.000} C_DIS
LIN {X -104.799,Y 223.903,Z 70.000,A 0.000,B 0.000,C 180.000,E1 0.000} C_DIS
LIN {X -116.185,Y 218.212,Z 70.000,A 0.000,B 0.000,C 180.000,E1 0.000} C_DIS
LIN {X -127.265,Y 211.941,Z 70.000,A 0.000,B 0.000,C 180.000,E1 0.000} C_DIS
LIN {X -138.007,Y 205.109,Z 70.000,A 0.000,B 0.000,C 180.000,E1 0.000} C_DIS
LIN {X -148.381,Y 197.734,Z 70.000,A 0.000,B 0.000,C 180.000,E1 0.000} C_DIS
LIN {X -158.364,Y 189.832,Z 70.000,A 0.000,B 0.000,C 180.000,E1 0.000} C_DIS
LIN {X -167.928,Y 181.427,Z 70.000,A 0.000,B 0.000,C 180.000,E1 0.000} C_DIS
LIN {X -177.044,Y 172.543,Z 70.000,A 0.000,B 0.000,C 180.000,E1 0.000} C_DIS
LIN {X -185.692,Y 163.200,Z 70.000,A 0.000,B 0.000,C 180.000,E1 0.000} C_DIS
LIN {X -189.755,Y 158.329,Z 70.000,A 0.000,B 0.000,C 180.000,E1 0.000} C_DIS
LIN {X 158.387,Y -189.812,Z 70.000,A 0.000,B 0.000,C 180.000,E1 0.000} C_DIS
LIN {X 158.364,Y -189.832,Z 70.000,A 0.000,B 0.000,C 180.000,E1 0.000} C_DIS
LIN {X 148.381,Y -197.734,Z 70.000,A 0.000,B 0.000,C 180.000,E1 0.000} C_DIS
LIN {X 138.007,Y -205.109,Z 70.000,A 0.000,B 0.000,C 180.000,E1 0.000} C_DIS
LIN {X 127.265,Y -211.941,Z 70.000,A 0.000,B 0.000,C 180.000,E1 0.000} C_DIS
LIN {X 116.185,Y -218.212,Z 70.000,A 0.000,B 0.000,C 180.000,E1 0.000} C_DIS
LIN {X 104.799,Y -223.903,Z 70.000,A 0.000,B 0.000,C 180.000,E1 0.000} C_DIS
LIN {X 93.132,Y -229.002,Z 70.000,A 0.000,B 0.000,C 180.000,E1 0.000} C_DIS
LIN {X 81.221,Y -233.493,Z 70.000,A 0.000,B 0.000,C 180.000,E1 0.000} C_DIS
LIN {X 69.094,Y -237.364,Z 70.000,A 0.000,B 0.000,C 180.000,E1 0.000} C_DIS
LIN {X 56.782,Y -240.606,Z 70.000,A 0.000,B 0.000,C 180.000,E1 0.000} C_DIS
LIN {X 52.994,Y -241.398,Z 70.000,A 0.000,B 0.000,C 180.000,E1 0.000} C_DIS
LIN {X -241.413,Y 53.009,Z 70.000,A 0.000,B 0.000,C 180.000,E1 0.000} C_DIS
LIN {X -241.988,Y 50.570,Z 70.000,A 0.000,B 0.000,C 180.000,E1 0.000} C_DIS
LIN {X -244.270,Y 38.044,Z 70.000,A 0.000,B 0.000,C 180.000,E1 0.000} C_DIS
LIN {X -245.906,Y 25.418,Z 70.000,A 0.000,B 0.000,C 180.000,E1 0.000} C_DIS
LIN {X -246.888,Y 12.728,Z 70.000,A 0.000,B 0.000,C 180.000,E1 0.000} C_DIS
LIN {X -247.215,Y 0.000,Z 70.000,A 0.000,B 0.000,C 180.000,E1 0.000} C_DIS
LIN {X -246.888,Y -12.728,Z 70.000,A 0.000,B 0.000,C 180.000,E1 0.000} C_DIS
LIN {X -245.906,Y -25.418,Z 70.000,A 0.000,B 0.000,C 180.000,E1 0.000} C_DIS
LIN {X -244.270,Y -38.044,Z 70.000,A 0.000,B 0.000,C 180.000,E1 0.000} C_DIS
LIN {X -241.988,Y -50.570,Z 70.000,A 0.000,B 0.000,C 180.000,E1 0.000} C_DIS
LIN {X -239.065,Y -62.957,Z 70.000,A 0.000,B 0.000,C 180.000,E1 0.000} C_DIS
LIN {X -235.506,Y -75.182,Z 70.000,A 0.000,B 0.000,C 180.000,E1 0.000} C_DIS
LIN {X -231.324,Y -87.206,Z 70.000,A 0.000,B 0.000,C 180.000,E1 0.000} C_DIS
LIN {X -226.528,Y -98.998,Z 70.000,A 0.000,B 0.000,C 180.000,E1 0.000} C_DIS
LIN {X -221.131,Y -110.529,Z 70.000,A 0.000,B 0.000,C 180.000,E1 0.000} C_DIS
LIN {X -215.148,Y -121.766,Z 70.000,A 0.000,B 0.000,C 180.000,E1 0.000} C_DIS
LIN {X -208.595,Y -132.679,Z 70.000,A 0.000,B 0.000,C 180.000,E1 0.000} C_DIS
LIN {X -201.488,Y -143.243,Z 70.000,A 0.000,B 0.000,C 180.000,E1 0.000} C_DIS
LIN {X -199.530,Y -145.851,Z 70.000,A 0.000,B 0.000,C 180.000,E1 0.000} C_DIS
LIN {X -145.843,Y -199.538,Z 70.000,A 0.000,B 0.000,C 180.000,E1 0.000} C_DIS
;rapid-leaky
$VEL.CP=0.3
LIN {X 77.682,Y 266.869,Z 80.000,A 0.000,B 0.000,C 180.000,E1 0.000} C_DIS
;bead-perimeter_outer
$VEL.CP=0.73
LIN {X 63.841,Y 270.513,Z 80.000,A 0.000,B 0.000,C 180.000,E1 0.000} C_DIS
LIN {X 49.830,Y 273.441,Z 80.000,A 0.000,B 0.000,C 180.000,E1 0.000} C_DIS
LIN {X 35.687,Y 275.644,Z 80.000,A 0.000,B 0.000,C 180.000,E1 0.000} C_DIS
LIN {X 21.451,Y 277.115,Z 80.000,A 0.000,B 0.000,C 180.000,E1 0.000} C_DIS
LIN {X 7.156,Y 277.853,Z 80.000,A 0.000,B 0.000,C 180.000,E1 0.000} C_DIS
LIN {X -7.156,Y 277.853,Z 80.000,A 0.000,B 0.000,C 180.000,E1 0.000} C_DIS
LIN {X -21.451,Y 277.115,Z 80.000,A 0.000,B 0.000,C 180.000,E1 0.000} C_DIS
LIN {X -35.687,Y 275.644,Z 80.000,A 0.000,B 0.000,C 180.000,E1 0.000} C_DIS
LIN {X -49.830,Y 273.441,Z 80.000,A 0.000,B 0.000,C 180.000,E1 0.000} C_DIS
LIN {X -63.841,Y 270.513,Z 80.000,A 0.000,B 0.000,C 180.000,E1 0.000} C_DIS
LIN {X -77.682,Y 266.869,Z 80.000,A 0.000,B 0.000,C 180.000,E1 0.000} C_DIS
LIN {X -91.317,Y 262.516,Z 80.000,A 0.000,B 0.000,C 180.000,E1 0.000} C_DIS
LIN {X -104.709,Y 257.467,Z 80.000,A 0.000,B 0.000,C 180.000,E1 0.000} C_DIS
LIN {X -117.825,Y 251.735,Z 80.000,A 0.000,B 0.000,C 180.000,E1 0.000} C_DIS
LIN {X -130.627,Y 245.336,Z 80.000,A 0.000,B 0.000,C 180.000,E1 0.000} C_DIS
LIN {X -143.084,Y 238.286,Z 80.000,A 0.000,B 0.000,C 180.000,E1 0.000} C_DIS
LIN {X -155.161,Y 230.604,Z 80.000,A 0.000,B 0.000,C 180.000,E1 0.000} C_DIS
LIN {X -166.826,Y 222.311,Z 80.000,A 0.000,B 0.000,C 180.000,E1 0.000} C_DIS
LIN {X -178.050,Y 213.428,Z 80.000,A 0.000,B 0.000,C 180.000,E1 0.000} C_DIS
LIN {X -188.801,Y 203.979,Z 80.000,A 0.000,B 0.000,C 180.000,E1 0.000} C_DIS
LIN {X -199.051,Y 193.990,Z 80.000,A 0.000,B 0.000,C 180.000,E1 0.000} C_DIS
LIN {X -208.773,Y 183.486,Z 80.000,A 0.000,B 0.000,C 180.000,E1 0.000} C_DIS
LIN {X -217.943,Y 172.495,Z 80.000,A 0.000,B 0.000,C 180.000,E1 0.000} C_DIS
LIN {X -226.533,Y 161.047,Z 80.000,A 0.000,B 0.000,C 180.000,E1 0.000} C_DIS
LIN {X -234.523,Y 149.172,Z 80.000,A 0.000,B 0.000,C 180.000,E1 0.000} C_DIS
LIN {X -241.892,Y 136.901,Z 80.000,A 0.000,B 0.000,C 180.000,E1 0.000} C_DIS
LIN {X -248.618,Y 124.268,Z 80.000,A 0.000,B 0.000,C 180.000,E1 0.000} C_DIS
LIN {X -254.686,Y 111.304,Z 80.000,A 0.000,B 0.000,C 180.000,E1 0.000} C_DIS
LIN {X -260.078,Y 98.045,Z 80.000,A 0.000,B 0.000,C 180.000,E1 0.000} C_DIS
LIN {X -264.780,Y 84.527,Z 80.000,A 0.000,B 0.000,C 180.000,E1 0.000} C_DIS
LIN {X -268.780,Y 70.785,Z 80.000,A 0.000,B 0.000,C 180.000,E1 0.000} C_DIS
LIN {X -272.067,Y 56.854,Z 80.000,A 0.000,B 0.000,C 180.000,E1 0.000} C_DIS
LIN {X -274.635,Y 42.773,Z 80.000,A 0.000,B 0.000,C 180.000,E1 0.000} C_DIS
LIN {X -276.472,Y 28.580,Z 80.000,A 0.000,B 0.000,C 180.000,E1 0.000} C_DIS
LIN {X -277.576,Y 14.309,Z 80.000,A 0.000,B 0.000,C 180.000,E1 0.000} C_DIS
